# B&R Automation Studio project JOB_NUMBER (part 5)

#### Kan_Driver.ab
```automation-basic
(********************************************************************
 * COPYRIGHT -- HP
 ********************************************************************
 * Program: Kan_Driver
 * File: Kan_Driver.ab
 * Author: treamsbottom
 * Created: September 07, 2012
 ********************************************************************
 * Implementation of program Kan_Driver
 ********************************************************************)
;----------------------------------------------------------------------------------------------------------------;
;-----21-1-2013..TR..Version A6 - First TestedVersion - Note 2 Specials in overview clien to run with Shuttle
;-----28-1-2013..TR..Version A7 - Remove Specials..Add option to send program and category number & Batch number.
;-----20-5-2014..TR..Version A12 - Fix ValidCat on DataValid
;-----09-01-2015..TR..Version A14 - Add Batching control
;-----02-08-2016 ..TR..Version A17 - Add Syncronous loading to Server Cmd 1000.. Use Comm[x].Transfer to watch for permission to unload.
;-----03-03-2017..TR.Version A18 - Add "Advanced Connection Mode"
;-----07-06-2017 ..TR..Version A19 - Fix issues with sending empty bag date-- Remove reference to Comm[].Category -- Read all information from bag for consistency.
;-----24-07-2018 ..TR -- Versioning Stopped Issues now tracked in GIT.
;-----------------------------------------------------------------------------------------------------------------
PROGRAM _INIT
	comm ACCESS ADR(Comm[0]);
END_PROGRAM
PROGRAM _CYCLIC
;Monitor State of supertrack (only send basic states now).
;IF (Kanlink.Server.Enable OR Kanlink.Client.Enable OR Kanlink.OverviewClient.Enable OR Kanlink.OverviewServer.Enable) THEN
;	IF SafetyZone[1].HaltSys THEN
;		SuperTrackState = KG_MACHINESTATE_EMERGENCYSTOP
;	ELSE
;		SuperTrackState = KG_MACHINESTATE_AUTOMATIC_RUN
;	ENDIF
;ENDIF
;--------------------------------------------------Kanlink Server Communication-----------------------------------------------------------------
IF Kanlink.Server.Enable THEN
	;Populate Batch Data
	LOOP n = 1 TO Kanlink.Server.MaxConns  DO
		IF (Kanlink.Server.IP[n].Adr > 0) THEN
			LOOP Index = 1 TO 1 DO ; Loop through each bag buffer
				comm ACCESS ADR(Comm[Kanlink.Server.IP[n].CommID]);
				IF (comm.Category > 0) THEN
					GetTimeStamp.enable = 1
					GetTimeStamp FUB DTGetTime()
					Batch[n].BatchData[Index].dtTimeStamp = GetTimeStamp.DT1
					;Make a string out OF CAT AND CUS
					length = itoa(comm.Category,ADR(myCategoryString));
					length = itoa(comm.Customer,ADR(myCustomerString));
					;copy Bag Data to KanLink Bag data type
;					IF Kanlink.GlobalSettings.TransferProgramCode THEN
;						Batch[n].BatchData[Index].sCategory = myProgramString
;						length = memcpy(ADR(Batch[n].BatchData[Index].bCustom),ADR(myCategoryString),12)
;					ELSE IF Kanlink.GlobalSettings.TransferProgin_bCustom THEN
;						Batch[n].BatchData[Index].sCategory = myCategoryString
;						length = memcpy(ADR(Batch[n].BatchData[Index].bCustom),ADR(myProgramString),12)
;					ELSE
						Batch[n].BatchData[Index].sCategory = myCategoryString
;					ENDIF
					IF Kanlink.GlobalSettings.UseBatchCode THEN
						IF Kanlink.GlobalSettings.BatchCodeTyp = BatchTyp_UDINT THEN
							;length = itoa(Bag[BagNumber].Mis,ADR(Batch[n].BatchData[Index].bBatchNo)) ; Convert to string
							length = memcpy(ADR(Batch[n].BatchData[Index].bBatchNo),ADR(comm.BatchID),4) ; Direct UDINT copy unreadble in KANLINK data.
						ELSE IF Kanlink.GlobalSettings.BatchCodeTyp = BatchTyp_16Byte THEN
							;Bag typ does not support this yet..
						ENDIF
					ELSE
						length = strcpy(ADR(Batch[n].BatchData[Index].bBatchNo),"")
					ENDIF
					Batch[n].BatchData[Index].bCntCustomers = 1
					Batch[n].BatchData[Index].wTotalWeight = comm.Weight;Summary weight of all Part Customers in the Bag, normally 1
					;First Customer in the Bag

					IF (comm.Batch_QtyRemaining <= 1) THEN
						Batch[n].BatchData[Index].PartBatch[0].sCustomNo = myCustomerString
						Batch[n].BatchData[Index].PartBatch[0].wCustomWeight = comm.Weight;Bag[BagNumber].Wgt
					ELSE
						Batch[n].BatchData[Index].bCntCustomers = USINT(comm.Batch_QtyRemaining)
						LOOP t = 0 TO 7 DO
							length = itoa(comm.Batchpart[t].Customer,ADR(myCustomerString));
							Batch[n].BatchData[Index].PartBatch[t].sCustomNo = myCustomerString
							Batch[n].BatchData[Index].PartBatch[t].wCustomWeight = comm.Batchpart[t].Wgt
						ENDLOOP
					ENDIF
				ELSE
					strcpy(ADR(myCategoryString),ADR(""));
					strcpy(ADR(myCustomerString),ADR(""))
					strcpy(ADR(myProgramString),ADR(""));
					Batch[n].BatchData[Index].bCntCustomers = 0
					Batch[n].BatchData[Index].sCategory = myCategoryString
					length = strcpy(ADR(Batch[n].BatchData[Index].bCustom),"")
					length = strcpy(ADR(Batch[n].BatchData[Index].bBatchNo),"")
					Batch[n].BatchData[Index].wTotalWeight = 0 ;Summaray weight of all Part Customers in the Bag, normally 1
					LOOP t = 0 TO 7 DO
						Batch[n].BatchData[Index].PartBatch[t].sCustomNo = myCustomerString
						Batch[n].BatchData[Index].PartBatch[t].wCustomWeight = 0
					ENDLOOP
				ENDIF
				PT100[n].Resp.BatchData = Batch[n].BatchData[1] ; Only send first bag over KANLINK
			ENDLOOP

			; Handshake Signal Convert Comm into the KANLINK protocol
			;ValidCat = 	strcmp(ADR(comm.Category), "")
			//BagNumber = Kanlink.Server.BagNum[n].BagNums[1];
			IF (comm.Category > 0) THEN
				PT100[n].Resp.xHsDataValid = TRUE;
			ELSE
				PT100[n].Resp.xHsDataValid = FALSE
				PT100[n].Resp.xHsUnloading = FALSE
			ENDIF

			IF comm.BagReady THEN
				PT100[n].Resp.xHsReqForUnload = TRUE;
			ELSE
				PT100[n].Resp.xHsReqForUnload = FALSE;
			ENDIF

			comm.ReadyToLoad	= PT100[n].Req.xHready;
			comm.DropLoad 		= PT100[n].Req.xHreadyForLoad;
			comm.LoadDropped  	= PT100[n].Req.xHbatchReceived;
			PT100[n].Resp.wCntLoads = comm.Batch_QtyRemaining

			IF comm.DropLoad THEN
				PT100[n].Resp.xHsUnloading = TRUE
			ENDIF

			IF comm.HaltSys THEN
				PT100[n].Resp.wState = KG_MACHINESTATE_EMERGENCYSTOP
			ELSE
				PT100[n].Resp.wState = KG_MACHINESTATEX_AUTOMATIC_RUN
			ENDIF

			comm.Live = IFhlKanLink.Server[n].out.xConnected
		;Syncronous Loading.
			IF PT100[n].Req.xHreqCtrlTransfer THEN
				//Syncronous loading. Only allow unload when bit .x.x.x. is on
				PT100[n].Resp.xHsTransferRunning := PT100[n].Req.xHwaitingForTransfer;
			ELSE
				//Always give permission to unload..
				PT100[n].Resp.xHsTransferRunning := 1;
			ENDIF;
			comm.Transfer := PT100[n].Resp.xHsTransferRunning
		ENDIF
	ENDLOOP
ENDIF//ServerDriver
;--------------------------------------------------------Client Driver------------------------------------------------------------------
IF Kanlink.Client.Enable THEN
	LOOP n = 1 TO Kanlink.Client.MaxConns DO
		comm  ACCESS ADR(Comm[Kanlink.Client.IP[n].CommID])
		;Give Machine Ready
		PTResp[n].Req.xHready = TRUE
		PTResp[n].Req.bHcmdAutomatic = TRUE

		comm.BagReady = PTResp[n].Resp.xHsReqForUnload
		;Give ready to load when Ready
		PTResp[n].Req.xHreadyForLoad = comm.ReadyToLoad
		PTResp[n].Req.xHtransferRunning = comm.Transfer

		PTResp[n].Req.xHbatchReceived = comm.LoadRecieved
			;Send supertrack state
		IF comm.HaltSys THEN
			PTResp[n].Req.wHstate = KG_MACHINESTATE_EMERGENCYSTOP
		ELSE
			PTResp[n].Req.wHstate = KG_MACHINESTATEX_AUTOMATIC_RUN
		ENDIF
		;Check for Data Valid and unloading start.	then copy data to Comm Variable
		UnloadingPulse[n].CLK = (PTResp[n].Resp.xHsUnloading AND PTResp[n].Resp.xHsDataValid)
		UnloadingPulse[n] FUB R_TRIG()
		IF UnloadingPulse[n].Q THEN
;			IF Kanlink.GlobalSettings.TransferProgramCode THEN
;				comm.Program = USINT(atoi(ADR(PTResp[n].Resp.BatchData.sCategory)))
;				comm.Category = atoi(ADR(PTResp[n].Resp.BatchData.bCustom))
;			ELSE IF Kanlink.GlobalSettings.TransferProgin_bCustom THEN
;				comm.Program = USINT(atoi(ADR(PTResp[n].Resp.BatchData.bCustom)))
;				comm.Category = atoi(ADR(PTResp[n].Resp.BatchData.sCategory))
;			ELSE
				comm.Category = atoi(ADR(PTResp[n].Resp.BatchData.sCategory))
;			ENDIF
			comm.Customer = atoi(ADR(PTResp[n].Resp.BatchData.PartBatch[0].sCustomNo))
			comm.Weight = PTResp[n].Resp.BatchData.wTotalWeight
			IF Kanlink.GlobalSettings.UseBatchCode THEN
				IF Kanlink.GlobalSettings.BatchCodeTyp = BatchTyp_UDINT THEN
					length = memcpy(ADR(comm.BatchID),ADR(PTResp[n].Resp.BatchData.bBatchNo),4)
				ELSE IF Kanlink.GlobalSettings.BatchCodeTyp = BatchTyp_16Byte THEN
					;Bag typ does not support this yet..
				ENDIF
			ELSE
				comm.BatchID = 0
			ENDIF
		ENDIF

		comm.Unloading =  PTResp[n].Resp.xHsUnloading
		UnloadingFinishPLS[n].CLK = PTResp[n].Resp.xHsUnloading
		UnloadingFinishPLS[n] FUB F_TRIG()

		comm.UnloadFinished = UnloadingFinishPLS[n].Q
		;Comm Live
		comm.Live = IFhlKanLink.Client[n].out.xConnected
	ENDLOOP
ENDIF
;;---------------------------------------------------------------------------------------------Overview Client----------------------------------------
;IF Kanlink.OverviewClient.Enable THEN ; Collect data
;;------------------------------------------Build Request---------------------------------------------------
;
;	LOOP n = 1 TO Kanlink.OverviewClient.MaxConns DO
;
;
;		IF (CANOffset > 0) THEN
;			CANOffset = (Kanlink.OverviewClient.CANOffset - 1)
;			Comm[n+CANOffset].Live = IFhlKanLink.Client[n+Kanlink.OverviewClient.IndexOffset].out.xConnected
;			IF NOT Comm[n+CANOffset].Live THEN
;				D[Kanlink.OverviewClient.StatusReg[n]] = 0
;			ENDIF
;		ELSE
;			CANOffset = 0
;		ENDIF;
;
;		IF Kanlink.OverviewClient.InfoReq[n].wNoOfPosition[6] = 0 THEN ; do not multiplex data.
;			STOverReq[n].Req.wCntPositions = Kanlink.OverviewClient.InfoReq[n].wCntPositions;Number of Bags requested
;			DataOffset[n] = 0
;		ELSE
;
;			DataCount = 0
;			LOOP x = 0 TO 5 DO
;				IF (STOverReq[n].Req.wNoOfPosition[x] > 0) THEN
;					DataCount = DataCount + 1
;				ENDIF
;				IF DataCount > 5 THEN
;					DataCount = 6
;				ENDIF
;			ENDLOOP
;			STOverReq[n].Req.wCntPositions = DataCount;Number of Bags requested
;		ENDIF
;
;
;		LOOP x = 0 TO 5 DO
;			;datapositions requested
;			EXITIF ((DataOffset[n] + x) > HLKANLINK_MAX_OVERVIEW_DATA)
;
;			STOverReq[n].Req.wNoOfPosition[x] = Kanlink.OverviewClient.InfoReq[n].wNoOfPosition[x + DataOffset[n]]
;				;-----------------------------------------------Read Data----------------------------------
;			IF (STOverReq[n].Resp.wNoOfPositions[x] > 0) AND ((x <= STOverReq[n].Resp.wCntPositions) OR (STOverReq[n].Resp.wCntPositions = 0 )) THEN
;				IF (Kanlink.OverviewClient.InfoResp[n].BagNum[x + DataOffset[n]] > 0) THEN
;					IF Kanlink.OverviewClient.InfoReq[n].wNoOfPosition[x+DataOffset[n]] = STOverReq[n].Resp.wNoOfPositions[x] THEN
;					//	D[Kanlink.OverviewClient.StatusReg[n]] = STOverReq[n].Resp.wMachineState
;						BagIndex = Kanlink.OverviewClient.InfoResp[n].BagNum[x + DataOffset[n]]
;						IF Kanlink.GlobalSettings.TransferProgramCode THEN
;							Bag[BagIndex].Prg = USINT(atoi(ADR(STOverReq[n].Resp.BatchData[x].sCategory)))
;							Bag[BagIndex].Cat = atoi(ADR(STOverReq[n].Resp.BatchData[x].bCustom))
;						ELSE IF Kanlink.GlobalSettings.TransferProgin_bCustom THEN
;							Bag[BagIndex].Prg = USINT(atoi(ADR(STOverReq[n].Resp.BatchData[x].bCustom)))
;							Bag[BagIndex].Cat = atoi(ADR(STOverReq[n].Resp.BatchData[x].sCategory))
;						ELSE
;							Bag[BagIndex].Cat = atoi(ADR(STOverReq[n].Resp.BatchData[x].sCategory))
;						ENDIF
;						Bag[BagIndex].Cus = atoi(ADR(STOverReq[n].Resp.BatchData[x].PartBatch[0].sCustomNo)) ; Standard line of code..
;						Bag[BagIndex].Wgt = STOverReq[n].Resp.BatchData[x].PartBatch[0].wCustomWeight
;						IF Kanlink.GlobalSettings.UseBatchCode THEN
;							IF Kanlink.GlobalSettings.BatchCodeTyp = BatchTyp_UDINT THEN
;									length = memcpy(ADR(Bag[BagIndex].Mis),ADR(STOverReq[n].Resp.BatchData[x].bBatchNo),4)
;								ELSE IF	Kanlink.GlobalSettings.BatchCodeTyp = BatchTyp_16Byte THEN
;								;Not supported yet....
;							ENDIF
;						ELSE
;							Bag[BagIndex].Mis = 0
;						ENDIF
;					ENDIF
;				ENDIF
;			ENDIF
;		ENDLOOP
;		IF STOverReq[n].Resp.wNoOfPositions[0] = Kanlink.OverviewClient.InfoReq[n].wNoOfPosition[DataOffset[n]] THEN
;			DataOffset[n] = DataOffset[n] + 6
;		ELSE IF Kanlink.OverviewClient.InfoReq[n].wNoOfPosition[DataOffset[n]] = 0 THEN
;			DataOffset[n] = 0
;		ENDIF
;	ENDLOOP
;ENDIF
;
;;---------------------------------------------------------------------------------------------Overview Server----------------------------------------
;IF Kanlink.OverviewServer.Enable THEN
;	LOOP n = 1 TO Kanlink.OverviewServer.MaxConns DO
;		IF (STOverResp[n].Req.wCntPositions <= 6) THEN
;			IF (STOverResp[n].Req.wCntPositions = 0) OR (STOverResp[n].Req.wCntPositions = 6) THEN
;				NoOfDataRequested = 5
;			ELSE
;				NoOfDataRequested = STOverResp[n].Req.wCntPositions
;			ENDIF
;			LOOP x = 0 TO 5 DO
;				IF x <= NoOfDataRequested THEN
;					BagIndex = STOverResp[n].Req.wNoOfPosition[x]
;
;					//STOverResp[n].Resp.wMachineState = SuperTrackState
;					STOverResp[n].Resp.wNoOfPositions[x] = BagIndex
;					STOverResp[n].Resp.wCntPositions = 	STOverResp[n].Req.wCntPositions
;					itoa(Bag[BagIndex].Prg,ADR(sProgram))
;					itoa(Bag[BagIndex].Cat,ADR(sCategory))
;					itoa(Bag[BagIndex].Cus,ADR(sCustomer))
;					itoa(Bag[BagIndex].Mis,ADR(sBatchID))
;					STOverResp[n].Resp.BatchData[x].dtTimeStamp = GetTimeStamp.DT1
;					IF Kanlink.GlobalSettings.TransferProgramCode THEN
;						strcpy(ADR(STOverResp[n].Resp.BatchData[x].sCategory),ADR(sProgram))
;						strcpy(ADR(STOverResp[n].Resp.BatchData[x].bCustom),ADR(sCategory))
;					ELSE IF Kanlink.GlobalSettings.TransferProgin_bCustom THEN
;						strcpy(ADR(STOverResp[n].Resp.BatchData[x].sCategory),ADR(sCategory))
;						strcpy(ADR(STOverResp[n].Resp.BatchData[x].bCustom),ADR(sProgram))
;					ELSE
;						strcpy(ADR(STOverResp[n].Resp.BatchData[x].sCategory),ADR(sCategory))
;					ENDIF
;					IF Kanlink.GlobalSettings.UseBatchCode THEN
;						IF Kanlink.GlobalSettings.BatchCodeTyp = BatchTyp_UDINT THEN
;							length = memcpy(ADR(STOverResp[n].Resp.BatchData[x].bBatchNo),ADR(Bag[BagIndex].Mis),4)
;						ELSE IF Kanlink.GlobalSettings.BatchCodeTyp = BatchTyp_UDINT THEN
;							strcpy(ADR(STOverResp[n].Resp.BatchData[x].bBatchNo),ADR(sBatchID))
;						ENDIF
;					ELSE
;						strcpy(ADR(STOverResp[n].Resp.BatchData[x].bBatchNo),"")
;					ENDIF
;					strcpy(ADR(STOverResp[n].Resp.BatchData[x].PartBatch[0].sCustomNo),ADR(sCustomer))
;					STOverResp[n].Resp.BatchData[x].PartBatch[0].wCustomWeight = Bag[BagIndex].Wgt
;				ELSE
;					STOverResp[n].Resp.wNoOfPositions[x] = 0
;					STOverResp[n].Resp.BatchData[x].dtTimeStamp = 0
;					strcpy(ADR(STOverResp[n].Resp.BatchData[x].sCategory),"")
;					strcpy(ADR(STOverResp[n].Resp.BatchData[x].bCustom),"")
;					strcpy(ADR(STOverResp[n].Resp.BatchData[x].bBatchNo),"")
;					strcpy(ADR(STOverResp[n].Resp.BatchData[x].PartBatch[0].sCustomNo),"")
;					STOverResp[n].Resp.BatchData[x].PartBatch[0].wCustomWeight = 0
;				ENDIF
;			ENDLOOP
;		ENDIF
;	ENDLOOP
;ENDIF

END_PROGRAM
```

### Package Logical/Standard/Kanlink/CAN - CAN Communication Variables

### CAN.typ
```iecst
TYPE
	WET_CAN : 	STRUCT
		ControlSignals : USINT;
		ControlSignals2 : USINT;
		Category : UINT;
		Customer : UINT;
		Weight : UINT;
	END_STRUCT;
	DRY_CAN : 	STRUCT
		ControlSignals : USINT;
		ControlByte2 : USINT;
		Category : UDINT;
		Weight : UINT;
	END_STRUCT;
	DRY_CAN1 : 	STRUCT
		CustomerCode : UDINT;
		BatchCode : UDINT;
	END_STRUCT;
	DRYCAN_comm_typ : 	STRUCT
		ReadFrame : DRY_CAN;
		WriteFrame : DRY_CAN;
		WriteFrame1 : DRY_CAN1;
		EventRead : BOOL;
		EventWrite : BOOL;
		EventWrite1 : BOOL;
	END_STRUCT;
	Comm_typ : 	STRUCT
		StrobeComplete : BOOL;
		BagReady : BOOL;
		BatchCode : UINT;
		Category : UDINT;
		Customer : UDINT;
		Destination : UINT;
		DropLoad : BOOL;
		DoubleLoad : BOOL;
		Live : BOOL;
		LiveTime : UINT;
		LoadDropped : BOOL;
		LoadFinished : BOOL;
		Program : UINT;
		ReadyToLoad : BOOL;
		UnloadFinished : BOOL;
		Weight : UINT;
		BatchID : UDINT;
		Batch_QtyRemaining : UINT;
		LoadRecieved : BOOL;
		Unloading : BOOL;
		Batchpart : ARRAY[0..7]OF Batchpart_typ;
		Batchpart_wgt : ARRAY[0..9]OF UINT;
		Count : UINT;
		Bid : UDINT; (**Internal use only pass bid ID>*)
		TimeStamp : DATE_AND_TIME; (**Internal use only*)
		Transfer : BOOL;
		HaltSys : BOOL;
	END_STRUCT;
	Batchpart_typ : 	STRUCT
		Wgt : UINT;
		Customer : UDINT;
	END_STRUCT;
END_TYPE
```

### CAN.var
```iecst
VAR CONSTANT
	MAX_COMM : USINT := 30;
END_VAR
VAR
	Comm : ARRAY[0..MAX_COMM] OF Comm_typ;
END_VAR
VAR CONSTANT
	COMM_CLEAR : Comm_typ := (0);
END_VAR
```

### Program Logical/Standard/Kanlink/kanlink_map (IEC) - *Custom task to convert Kanlink PLC to eVue Comms

#### Variables.var
```iecst
VAR
	bag_2_wieight : INT;
	doubleDrop : BOOL;
	DryerOpenTimer1 : TON;
	DryerOpenTimer2 : TON;
	DryerOpenTimer3 : TON;
	DryerOpenTimer4 : TON;
	DryerOpenTimer5 : TON;
	DryerOpenTimer6 : TON;
	DryerOpenTimer7 : TON;
	DryerOpenTimer8 : TON;
	DryerOpenTimer9 : TON;
	DryerOpenTimer10 : TON;
	DryerOpenTimer11 : TON;
	DryerOpenTimer12 : TON;
	DryerOpenTimer13 : TON;
	DryerOpenTimer14 : TON;
	DryerOpenTimer15 : TON;
	DryerOpenTimer16 : TON;
	WasherOpenTimer1 : TON;
	WasherOpenTimer2 : TON;
	WasherOpenTimer3 : TON;
	WasherOpenTimer4 : TON;
	WasherOpenTimer5 : TON;
	WasherOpenTimer6 : TON;
	WasherOpenTimer7 : TON;
	WasherOpenTimer8 : TON;
	WasherOpenTimer9 : TON;
	WasherOpenTimer10 : TON;
END_VAR
```

#### Cyclic.st
```iecst
PROGRAM _CYCLIC
//	//Opener code
//
//
//	//Tunnel X
//	r56.open_signal	:= 	Comm[1].DropLoad;
//	r56.receive_signal	:= 	Comm[1].LoadDropped;
//	Comm[1].BagReady	:= r56.sling_ready;
//
//	IF r56.sling_ready THEN
//		Comm[1].Customer	:= wash_com_cust_1;
//		Comm[1].Category	:= wash_com_cat_1;
//		Comm[1].BatchID		:= DByte_TO_4Byte(ADR(wash_com_batch1_1),ADR(wash_com_batch2_1));
//		Comm[1].Weight		:= (wash_com_wt_1 * 10);
//	ELSE
//		Comm[1].Customer	:= 0;
//		Comm[1].Category	:= 0;
//		Comm[1].BatchID		:= 0;
//		Comm[1].Weight		:= 0;
//	END_IF;
//
//	IF EDGEPOS(r56.fire) THEN
//		wash_com_cust_1 := 0;
//		wash_com_cat_1  := 0;
//		wash_com_wt_1  := 0;
//		wash_com_batch1_1 := 0;
//		wash_com_batch2_1 := 0;
//	END_IF;
//
//
//
//
//	//Washer X
//	WasherOpenTimer1(IN:= r60.sling_ready AND Comm[3].DropLoad, PT := t#1500ms);
//	IF EDGEPOS(Comm[3].ReadyToLoad) THEN
//		r60.transfer_requested_signal := TRUE;
//	END_IF;
//
//	r60.open_signal	:= 	WasherOpenTimer1.Q;
//	r60.receive_signal	:= 	Comm[3].LoadDropped;
//	Comm[3].BagReady	:= r60.sling_ready;
//
//
//	IF r60.sling_ready THEN
//		Comm[3].Customer	:= wash_com_cust_3;
//		Comm[3].Category	:= wash_com_cat_3;
//		Comm[3].BatchID		:= DByte_TO_4Byte(ADR(wash_com_batch1_3),ADR(wash_com_batch2_3));
//		Comm[3].Weight		:= (wash_com_wt_3 * 10);
//	ELSE
//		Comm[3].Customer	:= 0;
//		Comm[3].Category	:= 0;
//		Comm[3].BatchID		:= 0;
//		Comm[3].Weight		:= 0;
//	END_IF;
//
//	IF EDGEPOS(r60.fire) OR NOT(Comm[3].ReadyToLoad) THEN
//		r60.transfer_requested_signal := FALSE;
//	END_IF;
//
//	IF EDGEPOS(r60.fire) THEN
//		wash_com_cust_3 := 0;
//		wash_com_cat_3  := 0;
//		wash_com_wt_3  := 0;
//		wash_com_batch1_3 := 0;
//		wash_com_batch2_3 := 0;
//	END_IF;
//
//
//
//	//Dryer X
//	DryerOpenTimer1(IN:= r106.sling_ready AND Comm[6].DropLoad, PT := t#1500ms);
//	r106.transfer_requested_signal := Comm[6].ReadyToLoad;
//	r106.open_signal	:= 	DryerOpenTimer1.Q;
//	r106.receive_signal	:= 	Comm[6].LoadDropped;
//	Comm[6].BagReady	:= r106.sling_ready;
//
//	IF r106.sling_ready THEN
//		Comm[6].Customer	:= wash_com_cust_10;
//		Comm[6].Category	:= wash_com_cat_10;
//		Comm[6].BatchID		:= DByte_TO_4Byte(ADR(wash_com_batch1_10),ADR(wash_com_batch2_10));
//		Comm[6].Weight		:= (wash_com_wt_10 * 10);
//	ELSE
//		Comm[6].Customer	:= 0;
//		Comm[6].Category	:= 0;
//		Comm[6].BatchID		:= 0;
//		Comm[6].Weight		:= 0;
//	END_IF;
//
//	IF EDGEPOS(r106.fire) THEN
//		wash_com_cust_10 := 0;
//		wash_com_cat_10  := 0;
//		wash_com_wt_10  := 0;
//		wash_com_batch1_10 := 0;
//		wash_com_batch2_10 := 0;
//	END_IF;
//
//
//
//
//
//
//	// Transfers
//
//	//Wet Transfer X
//	wash_com_cust_6 	:= UDINT_TO_INT(Comm[28].Customer);
//	wash_com_cat_6 		:= UDINT_TO_INT(Comm[28].Category);
//	wash_com_wt_6 		:= (Comm[28].Weight/10);
//	wash_com_batch1_6	:= Get_Lower2Bytes(Comm[28].BatchID);
//	wash_com_batch2_6	:= Get_Higher2Bytes(Comm[28].BatchID);
//	//	Comm[28].bCustom[0]
//
//
//	Comm[28].ReadyToLoad	:= r80.sling_ready;
//	r80.transfer_requested_signal := Comm[28].BagReady;
//	r80.xfer_in_progress	:= Comm[28].Unloading;
//	r80.xfer_complete := Comm[28].UnloadFinished;
//
//	IF EDGEPOS(r80.fire) THEN
//		wash_com_cust_6 := 0;
//		wash_com_cat_6 := 0;
//		wash_com_wt_6 := 0;
//		wash_com_batch1_6 := 0;
//		wash_com_batch2_6 := 0;
//	END_IF;
END_PROGRAM
```

### Package Logical/Standard/Kanlink/KGFramework - Standard-Packages

### Package Logical/Standard/Kanlink/KGFramework/Pkg_KGStandard - Kannegiesser Standards

### Library Logical/Standard/Kanlink/KGFramework/Pkg_KGStandard/KGstdLib (IEC) - Kannegiesser Hilfsfunktionen
Depends on: astime, AsIODiag, Ethernet, AsBrStr, DataObj, AsArLog

#### kgGetEthPort.st - Returns the CPUs ethernet port as string
```iecst
(********************************************************************
* COPYRIGHT -- Microsoft
********************************************************************
* Library: Netlink
* File: GetEthPort.st
* Author: hunholz
* Created: June 30, 2011
********************************************************************
* Implementation of library Netlink
********************************************************************)

(* Returns the CPUs ethernet port as string *)
FUNCTION_BLOCK kgGetEthPort

IF enable THEN

	IF adrIF <= 16#3FFF THEN

		_bStep := 10;
		status := KG_ERR_GETETHPORT_ADRIF;
		RETURN;

	END_IF

	_xReady := FALSE;

	REPEAT

		CASE (_bStep) OF

			10:
				// Create Info
					DiagCreateInfo_CPU(enable := TRUE, infoKind := asdiagPLUGGED);

					status := DiagCreateInfo_CPU.status;

					IF (status = ERR_OK) THEN
			  			_bStep := 12;
					END_IF;

				12:
					// Get Info
					DiagGetNumInfo_CPU(enable := TRUE,
											ident := DiagCreateInfo_CPU.ident,
											index := 0,
											infoCode := asdiagPLUGGED_MODNO);

					status := DiagGetNumInfo_CPU.status;

					IF (status = ERR_OK) THEN

						CASE DiagGetNumInfo_CPU.value OF

							KG_CPU_X20CP1484, KG_CPU_X20CP1484_1, KG_CPU_X20CP3484_1, KG_CPU_X20CP1486, KG_CPU_X20CP3486, KG_CPU_X20CP3585, KG_CPU_X20CP1584,KG_CPU_X20CP1586, KG_CPU_X20CP3484:
								brsstrcpy(adrIF, ADR('IF2'));

							KG_CPU_PP420_1043_75, KG_CPU_CTT_11, KG_CPU_PP65_0571_P74, KG_CPU_PCT_04, KG_CPU_PCT_03:
								brsstrcpy(adrIF, ADR('IF5'));

							ELSE	// keinen gültigen B&R ID-Code gefunden
								brsstrcpy(adrIF, ADR('IF3'));
								//status := KG_ERR_GETETHPORT_IFSTRING;

						END_CASE

					_bStep := 14;

					ELSIF (status <> ERR_FUB_BUSY) THEN
						_bStep := 10;
				END_IF;

			14:
				 //Write string TO variable

				DiagDisposeInfo_CPU(enable := TRUE, ident := DiagCreateInfo_CPU.ident);

				status := DiagDisposeInfo_CPU.status;

				_xReady := (status = ERR_OK);

				IF (status <> ERR_FUB_BUSY) THEN

					_bStep := 10;
					DiagCreateInfo_CPU(enable := FALSE);
					DiagDisposeInfo_CPU(enable := FALSE);
					DiagGetNumInfo_CPU(enable := FALSE);

				END_IF;

			ELSE

				_bStep := 10;
				status := ERR_FUB_BUSY;

		END_CASE;

		UNTIL

		status <> ERR_OK OR _xReady

	END_REPEAT

ELSE

	status := ERR_FUB_ENABLE_FALSE;
	_bStep := 10;

END_IF

END_FUNCTION_BLOCK
```


- Program Logical/Standard/Kanlink/KGFramework/Pkg_mnSystem/mnSystem (IEC) - Systemtask für Versionierung (no source held here)

- Program Logical/Standard/Kanlink/KGFramework/Pkg_mnEth/mnEth (IEC) - Ethernetmanager (no source held here)

- Program Logical/Standard/Kanlink/KGFramework/Pkg_mnCnt/mnCnt (IEC) - Counter Manager (no source held here)

- Program Logical/Standard/Kanlink/KGFramework/Pkg_mnMsg/mnMsg (IEC) - Meldungsmanager (no source held here)

- Library Logical/Standard/Kanlink/KGFramework/Pkg_mnMsg/KGlibMsg (IEC) - A new source library (no source held here)

### Package Logical/Standard/Kanlink/KGFramework/Pkg_mnParam - Parameter-Manager

- Program Logical/Standard/Kanlink/KGFramework/Pkg_mnParam/mnParam (IEC) - Parameter Manager (no source held here)

### Library Logical/Standard/Kanlink/KGFramework/Pkg_mnParam/mnParamLib (IEC)
Depends on: astime


- Program Logical/Standard/Kanlink/KGFramework/Pkg_mnTxt/mnTxt (IEC) - Text-Manager (no source held here)

- Program Logical/Standard/Kanlink/KGFramework/Pkg_hlDFII/hlDFII (IEC) - Statemachine zur Abfrage einer SQL-Datenbank (no source held here)

- Program Logical/Standard/Kanlink/KGFramework/Pkg_mnTest/mnTest (IEC) - Testadapter (no source held here)

- Program Logical/Standard/Kanlink/KGFramework/Pkg_svCPCache/svCPCache (IEC) - Category-Program-Cache (no source held here)

### Program Logical/Standard/Kanlink/KGFramework/Pkg_hlKanLink/hlKanLink (IEC) - Kanlink Task

#### KanLinkCyclic.st - Cyclic code
```iecst
(********************************************************************
 * COPYRIGHT -- Herbert Kannegiesser GmbH
 ********************************************************************
 * Program: KanLink
 * File: KanLinkCyclic.st
 * Author: stahlhut
 * Created: December 23, 2011
 ********************************************************************
 * Implementation of program WetLink
 ********************************************************************)

(*

	Falls ohne Framework gearbeitet werden soll in den Eigenschaften der Task hlKanLink (Config. View Cpu.sw)
	im Tab. Compiler im Feld "Additional build options:" -D HLKANLINK_AUTONOM  eintragen
	Dazu das Package KanLinkAutonom importieren

*)

PROGRAM _CYCLIC

// Struktur für Visualisierung füllen

IFhlKL_Visu.out.iCycleTime := Kanlink._iCycleTime;
IFhlKL_Visu.out.step := Kanlink.Step;
IFhlKL_Visu.out.udNetId := Kanlink.udNetID;
IFhlKL_Visu.out.udpOpenStatus := Kanlink.udp.open.status;
IFhlKL_Visu.out.udpRecStatus := Kanlink.udp.rec.status;
IFhlKL_Visu.out.udpSendStatus := Kanlink.udp.send.status;
_wClt := LIMIT(0,IFhlKL_Visu.in.iCltNr,HLKANLINK_MAX_CLIENTCONNS);
  _wSrv := LIMIT(0,IFhlKL_Visu.in.iServerNr,HLKANLINK_MAX_SERVERCONNS);
IFhlKL_Visu.out.client := Kanlink.ClientListe[_wClt];
IFhlKL_Visu.out.server := Kanlink.ServerListe[_wSrv];

// Commando von der Visu verarbeiten
// Commando nur setzen wenn CmdResp = 0
// aufrufer muss nach ausführung cmdNr wieder auf 0 setzen!
IF IFhlKL_Visu.in.cmdNr <> IFhlKL_Visu.out.cmdResp THEN
	CASE IFhlKL_Visu.in.cmdNr OF
		0: IFhlKL_Visu.out.cmdResp := 0;
		1: // Neustart
			IFhlKL_Visu.out.cmdResp := 1;
			Kanlink.Step := 1;
		2: // Neustart mit lastId = 1
			Kanlink._uiLastId := 1;
			IFhlKL_Visu.out.cmdResp := 1;
			Kanlink.Step := 2;
		ELSE
			// unbekanntes Commando
			IFhlKL_Visu.out.cmdResp := 16#7FFF;

	END_CASE;
END_IF;

#ifndef HLKANLINK_AUTONOM // Logging nur mit kg-Framework

	// ===========================
	// Logging
	// ===========================

	IF _xRBReady THEN

		CASE _wLogStep OF

			0:
				_ReadRB(wPtrRead := _wPtrRBread, wPtrStart := _wPtrRBstart, wPtrWrite := _wPtrRBwrite);

				IF _ReadRB.wStatus = ERR_OK THEN

					CASE _LogEntry.wErrorNo OF

						0:
							_kgArLogWrite.text := 'OK';

						HLKANLINK_MSG_NO_STRUCDEF:

							_kgArLogWrite.text := 'Create Strucdefinition failed : {##AttrVar1} / {##AttrVar2}';
							_kgArLogWrite.var1 := _LogEntry.lAttr1;

						ELSE

							_kgArLogWrite.text := UINT_TO_STRING(_LogEntry.wErrorNo);
							_kgArLogWrite.text := CONCAT(_kgArLogWrite.text, ' : {##AttrVar1} / {##AttrVar2}');
							_kgArLogWrite.var1 := _LogEntry.lAttr1;
							_kgArLogWrite.var2 := _LogEntry.lAttr2;

					END_CASE

					_wLogStep := 1;

				END_IF

			1:
				_kgArLogWrite();

				IF _kgArLogWrite.status <> ERR_FUB_BUSY THEN

					_wLogStep := 0;

				END_IF

		END_CASE

	END_IF

	IF _wDebIdx >= 0 AND _wDebIdx <= _HLKANLINK_MAX_IDX_DEFSTRUC THEN

		IF _lPtrStrucDef[_wDebIdx] > 0 THEN

			_sDebString ACCESS _lPtrStrucDef[_wDebIdx] + _wDebOffset;

		END_IF

	END_IF

#endif

	// =======================================================================

	IF _xInitOK THEN

		IF _xSaveConfig THEN
			KL_SaveConfDO_0(adrName :=ADR('KL_Conf') , adrDaten := ADR(IFhlKanLink.Parameter), len := SIZEOF( IFhlKanLink.Parameter));
			IF KL_SaveConfDO_0.status <> ERR_FUB_BUSY THEN // fertig
				_xSaveConfig := FALSE;
			END_IF;
		END_IF;

		IF EDGEPOS(IFhlKanLink.in.xRun ) THEN
			IF Kanlink.Step = 0 THEN
				Kanlink.Step := 1;
			END_IF;
		END_IF;
		IF EDGENEG(IFhlKanLink.in.xRun) THEN // stoppen
			IF Kanlink.Step <> 0 THEN
				Kanlink.Step := 20;
			END_IF;
		END_IF;

		IF IFhlKanLink.in.xRestart THEN
			Kanlink.Step := 1;
			IFhlKanLink.in.xRestart := 0;
		END_IF;

		IFhlKanLink.xError := (Kanlink.Step = 200);

		CASE Kanlink.Step OF

			0: //nix tun

			100: // Error nr in Logger eintragen

				Kanlink.Step := 200;

			200: // Auf User warten

			1: // init

				Kanlink.KLLib_Init_0(enable := 1, adrServer := ADR(Kanlink),adrInterface := ADR(IFhlKanLink));
				IF Kanlink.KLLib_Init_0.status = ERR_OK THEN
					Kanlink.Step := 10;
				ELSIF Kanlink.KLLib_Init_0.status <> ERR_FUB_BUSY THEN // fehler
					WL_ErrorNr := 10;
					Kanlink.Step := 100;

					IF _xRBReady THEN

						_LogEntryIn.wErrorNo := 10;
						_InsertRB(wPtrStart := _wPtrRBstart, wPtrRead := _wPtrRBread, wPtrWrite := _wPtrRBwrite);

					END_IF

				END_IF;

			10: // Kanlink Run

			20: // Kanlink schliessen

				Kanlink.udp.close.enable := 1;
				Kanlink.udp.close.ident := Kanlink._uiLastId;
				Kanlink.udp.close;
				IF Kanlink.udp.close.status = 0 THEN
					Kanlink.Step := 0;
				ELSIF Kanlink.udp.close.status = ERR_FUB_BUSY THEN

				ELSE
					Kanlink.Step := 100;
				END_IF;

		END_CASE;

		// interne Zustände auf out Struktur legen
		IFhlKanLink.out.iStep  := Kanlink.Step;
		// noch auzufüllen ....
//		IFhlKanLink.out.iError := ??;
//		IFhlKanLink.out.iClientError[0] := ??;
//		IFhlKanLink.out.iServerError[0] := ??;

		// hier beenden wenn zyklus nicht erlaubt
		IF  Kanlink.Step <> 10 THEN
			RETURN;
		END_IF;

		Kanlink;

		// falls Kanlink nix zu tun hat, hier beenden
		IF Kanlink.xReturn THEN
			RETURN;
		END_IF;

		// ------------------------------------------------------------------
		// Falls ein Request eines Clients aufgelaufen ist

		IF Kanlink._xGetServerReq THEN  // Req eines Clients angenommen, bearbeiten

			actGetServerReq;

			Kanlink._xGetServerReq := FALSE;
			Kanlink.udp.rec.enable := 1;

			RETURN;  // Daten sind versendet. Also Ende.

		END_IF;

		// ------------------------------------------------------------------------------
		// falls Response von einem Request kommt:

		IF Kanlink._xGetClientResp THEN // Response auf ClientReq angekommen
			actResponse;

		END_IF;

		// ------------------------------------------------------------------------------
		// Überprüfen ob per Hand bearbeitete Requests versendet werden müssen..

		IF  Kanlink.udp.send.enable = 0 THEN
			_xServerFound := 0;

			FOR _i:=0 TO HLKANLINK_MAX_SERVERCONNS  DO
				_ptrIndex ACCESS ADR(Kanlink.ServerListe[_iLastServerIdx]);
				_dSrvIf ACCESS _ptrIndex.adrInterface;
				IF (_ptrIndex.xReqManually AND (_dSrvIf.iState = 2)) THEN
					_xServerFound := 1;

					_iLastServerIdx := _iLastServerIdx + 1; // testen
					IF _iLastCltIdx > HLKANLINK_MAX_SERVERCONNS THEN
						_iLastServerIdx := 0;
					END_IF;
					EXIT;
					END_IF;
					_iLastServerIdx := _iLastServerIdx + 1; // testen
					IF _iLastServerIdx > HLKANLINK_MAX_SERVERCONNS THEN
					_iLastServerIdx := 0;
				END_IF;

			END_FOR;

			IF _xServerFound THEN
				Kanlink.ServerData.HeaderV1Send[0].Command := _ptrIndex.Cmd + 1;
				Kanlink.ServerData.HeaderV1Send[0].dataFormat := 5;
				Kanlink.ServerData.HeaderV1Send[0].Length := UDINT_TO_UINT( _ptrIndex.RespLength);
				Kanlink.ServerData.HeaderV1Send[0].ReqID := _ptrIndex.iReqID;
				Kanlink.ServerData.HeaderV1Send[0].CmdNr := _ptrIndex.CmdOpt AND 16#00FF;
				_ptrIndex.iConnectionTimer := 0;
				KLLib_SendData(ADR(Kanlink),_ptrIndex.AdrDataResp,_ptrIndex.RespLength,ADR(_ptrIndex.sClientIPAdr),-1,-1,0);
				_dSrvIf.iState := 0;
				RETURN;
			END_IF;
		END_IF;

		IF Kanlink._xSendClient THEN  // hier den Clienten bearbeiten
			_xCltFound := FALSE;
			_iCltIdx := -1;
			_iMuCltIdx := -1;

			FOR _i:=0 TO HLKANLINK_MAX_CLIENTCONNS  DO
				IF (Kanlink.ClientListe[_iLastCltIdx].MuClient >= 0) THEN
					IF ((Kanlink.MuClientListe[Kanlink.ClientListe[_iLastCltIdx].MuClient].bUse = 0) OR (Kanlink.MuClientListe[Kanlink.ClientListe[_iLastCltIdx].MuClient].bUse = 255)) THEN
						_xCheckClt := TRUE;
					ELSE
						_xCheckClt := FALSE;
					END_IF
				ELSE
					_xCheckClt := TRUE;
				END_IF

				IF (_xCheckClt = TRUE) THEN
					_dClient ACCESS ADR(Kanlink.ClientListe[_iLastCltIdx]);
					IF _dClient.adrInterface <> 0 THEN
						_dCltIf ACCESS _dClient.adrInterface;
					ELSE
						_dCltIf ACCESS ADR(_ifDummy);
					END_IF;
						// gefunden wenn kein ReqPend, Commando <> 0 todo gültige Adresse etc...
					IF _dClient.iCycleTime = 0 THEN
						_xSendNow := (_dCltIf.iState = 1) OR (_dCltIf.iState = 4) ; // falls angetickt oder timeout
					ELSE
						_xSendNow := (_dClient.iCycleWait > _dClient.iCycleTime);
					END_IF;
					IF 	(NOT _dClient.xReqPending) AND (_dClient.Cmd <> 0) AND _dClient.xActiv AND (_xSendNow) THEN
			  			_xCltFound := TRUE;
						_iCltIdx := _iLastCltIdx;
						_iLastCltIdx := _iLastCltIdx + 1; // testen
						IF _iLastCltIdx > HLKANLINK_MAX_CLIENTCONNS THEN
				  			_iLastCltIdx := 0;
						END_IF;
						EXIT;
					END_IF;
				END_IF

				_iLastCltIdx := _iLastCltIdx + 1; // testen
				IF _iLastCltIdx > HLKANLINK_MAX_CLIENTCONNS THEN
		  			_iLastCltIdx := 0;
				END_IF;

			END_FOR;

			IF (NOT _xCltFound) THEN
				FOR _i:=0 TO HLKANLINK_MAX_MU_CLIENTCONNS DO
					IF ((Kanlink.MuClientListe[_iLastMuCltIdx].bUse = 1) OR (Kanlink.MuClientListe[_iLastMuCltIdx].bUse = 2)) THEN

						IF Kanlink.ClientListe[Kanlink.MuClientListe[_iLastMuCltIdx].Clients[0]].adrInterface <> 0 THEN
							_dCltIf ACCESS Kanlink.ClientListe[Kanlink.MuClientListe[_iLastMuCltIdx].Clients[0]].adrInterface;
						ELSE
							_dCltIf ACCESS ADR(_ifDummy);
						END_IF;
							// gefunden wenn kein ReqPend, Commando <> 0 todo gültige Adresse etc...
						IF Kanlink.MuClientListe[_iLastMuCltIdx].iCycleTime = 0 THEN
							_xSendNow := (_dCltIf.iState = 1) OR (_dCltIf.iState = 4) ; // falls angetickt oder timeout
						ELSE
							_xSendNow := (Kanlink.MuClientListe[_iLastMuCltIdx].iCycleWait > Kanlink.MuClientListe[_iLastMuCltIdx].iCycleTime);
						END_IF;

						IF 	(NOT Kanlink.MuClientListe[_iLastMuCltIdx].xReqPending) AND Kanlink.MuClientListe[_iLastMuCltIdx].xActiv AND (_xSendNow) THEN
				  			_xCltFound := TRUE;
							_iMuCltIdx := _iLastMuCltIdx;
							_iLastMuCltIdx := _iLastMuCltIdx + 1; // testen
							IF _iLastMuCltIdx > HLKANLINK_MAX_MU_CLIENTCONNS THEN
					  			_iLastMuCltIdx := 0;
							END_IF;
							EXIT;
						END_IF;

					END_IF

					_iLastMuCltIdx := _iLastMuCltIdx + 1; // testen
					IF _iLastMuCltIdx > HLKANLINK_MAX_MU_CLIENTCONNS THEN
			  			_iLastMuCltIdx := 0;
					END_IF;

				END_FOR;
			END_IF

			IF NOT _xCltFound THEN
				Kanlink._xSendClient := FALSE;
				RETURN;

			ELSE

				IF (_iCltIdx >= 0) THEN
					// Client gefunden
					_dClient.iCnt := _dClient.iCnt + 1 ;
					_dClient.iReqId := _dClient.iReqId +1;
					_dClient.TimeOutLeft := _dClient.TimeOut;

					IF _dCltIf.iState = 1 THEN // falls über state dann "schnellwiederholung" aktivieren
						_dClient.iTimeOutCnt := 0; // scharf machen für den nächsten versuch
					END_IF;
					_dCltIf.iState := 2;

					Kanlink.ServerData.HeaderV1Send[0].Command := _dClient.Cmd;
					Kanlink.ServerData.HeaderV1Send[0].CmdNr := _dClient.CmdOpt AND 16#00FF;

					Kanlink.ServerData.HeaderV1Send[0].dataFormat := 5;
					Kanlink.ServerData.HeaderV1Send[0].Length := UDINT_TO_UINT( _dClient.ReqLength);
					Kanlink.ServerData.HeaderV1Send[0].ReqID := _dClient.iReqId;
					Kanlink.ServerData.HeaderV1Send[0].Tag		:= _dCltIf.tag;

// warum ?			KLLib_SendData(ADR(Kanlink),0,                  0,                 ADR(_dClient.sClientAdr),_iCltIdx,-1,KLLIB_REQ);
					KLLib_SendData(ADR(Kanlink),_dClient.AdrDataReq,_dClient.ReqLength,ADR(_dClient.sClientAdr),-1,      -1,KLLIB_REQ);

					_dClient.xReqPending := TRUE;
					_dClient.iCycleWait := 0;

					Kanlink._xSendClient := FALSE;

					RETURN;

				ELSIF (_iMuCltIdx >= 0) THEN

					// Client gefunden
					Kanlink.MuClientListe[_iMuCltIdx].iCnt := Kanlink.MuClientListe[_iMuCltIdx].iCnt + 1;
					Kanlink.MuClientListe[_iMuCltIdx].iReqId := Kanlink.MuClientListe[_iMuCltIdx].iReqId + 1;
					Kanlink.MuClientListe[_iMuCltIdx].TimeOutLeft := Kanlink.MuClientListe[_iMuCltIdx].TimeOut;

					IF _dCltIf.iState = 1 THEN // falls über state dann "schnellwiederholung" aktivieren
						Kanlink.MuClientListe[_iMuCltIdx].iTimeOutCnt := 0; // scharf machen für den nächsten versuch
					END_IF;
					_dCltIf.iState := 2;

					FOR _i := 0 TO KLLIB_MAX_MUL DO

						IF (Kanlink.MuClientListe[_iMuCltIdx].Clients[_i] >= 0) THEN

							Kanlink.ClientListe[Kanlink.MuClientListe[_iMuCltIdx].Clients[_i]].iCnt := Kanlink.MuClientListe[_iMuCltIdx].iCnt;
							Kanlink.ClientListe[Kanlink.MuClientListe[_iMuCltIdx].Clients[_i]].iReqId := Kanlink.MuClientListe[_iMuCltIdx].iReqId;
							Kanlink.ClientListe[Kanlink.MuClientListe[_iMuCltIdx].Clients[_i]].TimeOutLeft := Kanlink.MuClientListe[_iMuCltIdx].TimeOut;

							Kanlink.ServerData.HeaderV1Send[_i].Command := Kanlink.ClientListe[Kanlink.MuClientListe[_iMuCltIdx].Clients[_i]].Cmd;
							Kanlink.ServerData.HeaderV1Send[_i].CmdNr := Kanlink.ClientListe[Kanlink.MuClientListe[_iMuCltIdx].Clients[_i]].CmdOpt AND 16#00FF;

							Kanlink.ServerData.HeaderV1Send[_i].dataFormat := 5;
							Kanlink.ServerData.HeaderV1Send[_i].Length := UDINT_TO_UINT(Kanlink.ClientListe[Kanlink.MuClientListe[_iMuCltIdx].Clients[_i]].ReqLength);
							Kanlink.ServerData.HeaderV1Send[_i].ReqID := Kanlink.ClientListe[Kanlink.MuClientListe[_iMuCltIdx].Clients[_i]].iReqId;
							Kanlink.ServerData.HeaderV1Send[_i].Tag	:= _dCltIf.tag;

						END_IF

					END_FOR

					KLLib_SendData(ADR(Kanlink),0,0,ADR(Kanlink.MuClientListe[_iMuCltIdx].sClientAdr),-1,_iMuCltIdx,KLLIB_REQ);

					Kanlink.MuClientListe[_iMuCltIdx].xReqPending := TRUE;
					Kanlink.MuClientListe[_iMuCltIdx].iCycleWait := 0;

					FOR _i := 0 TO KLLIB_MAX_MUL DO

						IF (Kanlink.MuClientListe[_iMuCltIdx].Clients[_i] >= 0) THEN

							Kanlink.ClientListe[Kanlink.MuClientListe[_iMuCltIdx].Clients[_i]].xReqPending := TRUE;
							Kanlink.ClientListe[Kanlink.MuClientListe[_iMuCltIdx].Clients[_i]].iCycleWait := 0;
						END_IF

					END_FOR

					Kanlink._xSendClient := FALSE;

					RETURN;

				END_IF

			END_IF;

		END_IF;	// sendClient

#ifndef  HLKANLINK_AUTONOM  // wird MIT Framework gearbeitet
	ELSIF IFmnParam.Out.xParamOK AND IFmnEth.Out.xDataValid THEN

		Kanlink.ServerData.MetaInfoResp.KanLink_Hostname := IFmnEth.Out.IP.sHostname;
		Kanlink.ServerData.MetaInfoResp.Machine_type := WSTRING_TO_STRING(IFmnParam.Out.HeaderVersion.utfMachineType);
		Kanlink.ServerData.MetaInfoResp.DataModelTimeStamp := IFmnParam.Out.HeaderVersion.dtTimestamp;
		Kanlink.ServerData.MetaInfoResp.DataModelVersion := IFmnParam.Out.HeaderVersion.wVersion;

		Kanlink.ServerData.PingResp.KanLink_Hostname := IFmnEth.Out.IP.sHostname;

		_xInitOK := TRUE;

	END_IF
#else  // falls OHNE Framework gearbeitet wird
	ELSIF TRUE THEN
		_xInitOK := TRUE;
	END_IF
#endif

END_PROGRAM

PROGRAM _EXIT

	Kanlink.udp.close.enable	:= TRUE;
	Kanlink.udp.close.ident		:= Kanlink.udp.open.ident;
	Kanlink.udp.close;

END_PROGRAM
```

### Library Logical/Standard/Kanlink/KGFramework/Pkg_hlKanLink/KanLinkLib (IEC, version 0.94.5) - KanlinkHilfsfunktionen
Depends on: AsUDP, asstring, AsARCfg, brsystem, sys_lib, AsArLog, AsIODiag, AsETH, DataObj, KL_UserLib, KGstdLib

### KGFramework.ReleaseNotes.txt
```
0.08.0	2012-06-04	- mnParam Version 0.23.0. Siehe history.Pkg_mnParam.txt
					- mnSystem Version 1.04.0. Siehe mnSystem.History.txt
0.09.0	2012-06-12	- mnParam Version 0.24.0. Siehe history.Pkg_mnParam.txt
					- KGStandard Version 1.21.0
					- mnSystem Version 1.05.0
					- svCPCache Version 0.03.0
					- hlDFII Version 1.17.0. ACHTUNG: Parameterstruktur hat sich verändert!!!
0.10.0	2012-06-25	- KGStandar Version 1.22.0
					- mnSystem Version 1.06.0
					- mnParam Version 0.24.1
					- svCPCache Version 0.03.1
0.11.0	2012-07-03	- KGStandard Version 1.23.0
					- mnSystem Version 1.07.0
					- mnMsg Version 1.12.0 - Bugfix
					- mnParam Version 0.24.2 - Bugfix
					- svCPCache Version 0.03.2 - Bugfix
					- mnEth Version 2.10.1 - Bugfix
0.12.0	2012-07-18	- KGStandard Version 1.24.0
0.12.1	2012-08-30	- hlKanLink 0.94.4 - Bugfix
0.12.2	2012-09-03	- mnParam 0.24.3 - Bugfixes
0.13.0	2012-09-04	- mnTxt 0.09.0
					- mnParam 0.25.0
0.14.0	2012-09-05	- mnSystem 1.08.0
					- KGStandard 1.25.0
```

### Package Logical/Standard/Kanlink/KGFrameworkShare - Benutzereinstellungen


### Package Logical/Standard/Kanlink/KGFrameworkShare/Pkg_hlKanLinkUser - Kanlink User

### Library Logical/Standard/Kanlink/KGFrameworkShare/Pkg_hlKanLinkUser/KL_UserLib (IEC, version 0.91.0) - Kanlink User Library

#### KL_UserLib.var - Exported constants
```iecst
(********************************************************************
 * COPYRIGHT -- Herbert Kannegiesser GmbH
 ********************************************************************
 * Library: WL_UserLib
 * File: WL_UserLib.var
 * Author: stahlhut
 * Created: January 10, 2012
 ********************************************************************
 * Constants of library WL_UserLib
 ********************************************************************)
VAR CONSTANT
	HLKANLINK_MAX_CLIENTCONNS : UINT := 10; (*Anzahl der Clienten *)
	HLKANLINK_MAX_SERVERCONNS : UINT := 20; (*Anzahl der Server *)
	HLKANLINK_MAX_MU_CLIENTCONNS : UINT := 5;
	HLKANLINK_MAX_OVERVIEW_DATA : UINT := 35; (*Maximum data transfer on 1 overview connections*)
END_VAR
```


- Library Logical/Standard/Kanlink/KGFrameworkShare/Pkg_mnTestUser/libTestUse (IEC) - Userlibrary für Testadapter (no source held here)

- Program Logical/Standard/Kanlink/KGFrameworkShare/Pkg_mnTestUser/mnTestUser (IEC) - Initialisierung des Test (no source held here)

### Program Logical/Standard/Safety/AccessControl (IEC) - *Mapping to allow access into zones

#### Variables.var
```iecst
VAR
	n : INT;
END_VAR
```

#### Main.st
```iecst
PROGRAM _CYCLIC

//	Std.SafetyOnZone[1]	;High level
//	Std.SafetyOnZone[2]	;Maintenance platform
//	Std.SafetyOnZone[3]	;Low level
//	Std.SafetyOnZone[4]	;Belt load SL's
//	Std.SafetyOnZone[5]	;SSL3
//No access on zone 0

//	SafetyZone[0].BagsInTransit :=  FALSE;  // Safe to enter when false (Switch is NO) FALSE WHEN OK..
//	SafetyZone[0].HoistsOutOfPosition := FALSE; //<-- This is used to stop the door from opening if not position FALSE IS OK -- SWITCH IS NC..

	FOR n := 1 TO MAX_SAFE_ZONES DO
		SafetyZone[n].BagsInTransit :=  FALSE;
	//	SafetyZone[n].HoistsOutOfPosition := Hoist_Safety[n].OutOfPosition;
	END_FOR;

END_PROGRAM
```

### Program Logical/Standard/Safety/Safety (IEC)

#### Variables.var
```iecst
VAR CONSTANT
	MAX_SAFE_SYSTEMS : USINT := 1; (*Number of independant safety systems*)
END_VAR
VAR
	n : UINT;
	transitSettlePT : UDINT; (*Determines the amount of time to wait for bags in transit to settle before opening the interlock*)
	ton_10ms_Transit_Settle : ARRAY[0..MAX_SAFE_ZONES] OF TON_10ms; (*Determines the amount of time to wait for bags in transit to settle before opening the interlock*)
	safeState : ARRAY[0..MAX_SAFE_ZONES] OF USINT; (*USINT that tracks the state of the safe system so it can control the tower light*)
	debounceMasterPT : UDINT;
	masterReset : ARRAY[0..MAX_SAFE_ZONES] OF BOOL;
	ton_10ms_Master_Reset : ARRAY[0..MAX_SAFE_SYSTEMS] OF TON_10ms;
	masterResetRequest : ARRAY[0..MAX_SAFE_SYSTEMS] OF BOOL;
	startUpWarningPT : UDINT;
	ton_10ms_startUp_Warning : ARRAY[0..MAX_SAFE_SYSTEMS] OF TON_10ms;
	tp_10ms_reset_Pulse : TP_10ms;
	enableMasterReset : ARRAY[0..MAX_SAFE_SYSTEMS] OF BOOL;
	ton_10ms_Reset_Debounce : ARRAY[0..MAX_SAFE_ZONES] OF TON_10ms;
	ton_10ms_bagsInTransit : ARRAY[0..MAX_SAFE_ZONES] OF TON_10ms;
	f_trigRequestAccess : ARRAY[0..MAX_SAFE_ZONES] OF F_TRIG;
	ton_entryError : ARRAY[0..MAX_SAFE_ZONES] OF TON_10ms;
	resetRequired : ARRAY[0..MAX_SAFE_SYSTEMS] OF BOOL;
	lockDoor : ARRAY[0..MAX_SAFE_ZONES] OF BOOL;
	tof_HoistsOutOfPosition : ARRAY[0..MAX_SAFE_ZONES] OF TOF_10ms;
	safeZone : REFERENCE TO SafeZoneType;
	startZone : ARRAY[0..MAX_SAFE_SYSTEMS] OF UINT;
	endZone : ARRAY[0..MAX_SAFE_SYSTEMS] OF UINT;
	s : USINT;
	masterZone : BOOL;
	alarmCondition : ARRAY[0..MAX_SAFE_SYSTEMS] OF BOOL;
	tmrAlmOutput : ARRAY[0..MAX_SAFE_SYSTEMS] OF TON;
	masterZoneNo : UINT;
	safe2 : REFERENCE TO SafeZoneType;
END_VAR
```

#### _decodeData.st
```iecst
ACTION _decodeData:

//	Zone Status Encoding
//	0 - Zone Input State
//	1 - Zone Ready FOR Reset
//	2 - E-stop FUB error
//	3 - EDM Input State
//	4 - EDM Ready
//	5 - EDM Error
//	6 - EDM Disabled
//	7 - Zone Dependancy
//	8 - Safe System OK
//	9 - Auto Reset
//	10 - ACCESS Request
//	11 - Zone Status

safeZone.SafeInput				:= safeZone.DataFromSafePLC.0;
safeZone.Zone_Status 			:= safeZone.DataFromSafePLC.11;
safeZone.ResetReady				:= safeZone.DataFromSafePLC.1;
safeZone.RequestAccess		:= safeZone.DataFromSafePLC.10;   // Derived in the PLC from from Zone Healthy and Reset Push button

END_ACTION
```

#### Main.st
```iecst
//---------------------------------------------
//-------------Safety Request------------------
//---------------------------------------------
//V1.00.2 -- 2019 May 24 -- TR -- Fix issue with master reset not working if not ready.
//V1.00.3 -- 2019 June 26 -- TR -- FIx issue with the solenoid not opening if the hoist switch is made after the bagInTransit timers.. Add timer for hoist in position so the hoist cannot be moving past the safe position and open the door.
//V1.00.4 -- 2019 November 11 -- TR -- 	FIX: Issues with the solenoid locking incorrectly,
						//ADD: Control to lift the edge protection gates ( Map Directly to all required outputs.)
//V1.00.5 -- 2020 Decemeber 16 -- TR -- UPDATE : Change to new structure for Safety.
//V1.00.6 -- 2021 January 02 -- TR -- UPDATE : Add Test Mode bit
//V2.00.1 - 2001 Feburary 05 - Change Structures to remove links to direct IO points. Data now comes from Safe PLC.

PROGRAM _INIT

//***************************************************************************************
//	N.B Zone 11 has been faked so we can control the lamp tower correctly FOR the primary
//***************************************************************************************

//DECLARE MAX_SAFE_SYSTEMS IN CONTSTANTS

	startZone[1] := 1;   // Number of the Master Zone
	endZone[1] := 6;	// Last zone in the area
	enableMasterReset[1] := TRUE; // Set to true if master reset is to be used/
//	alarmCondition[1] := system_alarm_1 OR soiled_validation_alarm OR halted;

//	//zone for clean alarms.
//	startZone[2] := 11;   // Number of the Master Zone
//	endZone[2] := MAX_SAFE_ZONES;	// Last zone in the area
//	enableMasterReset[2] := TRUE; // Set to true if master reset is to be used/

	//NB//  A ZONE CANNOT BELONG TO MORE THAN 1 SAFE SYSTEM.

	// MAX Zone if 30

	debounceMasterPT := 476; //4.76 second
	transitSettlePT := 3000; //3000seconds
	startUpWarningPT := 500; //5 secs

	FOR n:=1 TO MAX_SAFE_ZONES DO
		safeState[n] := 4;
	END_FOR;

	#if (MAX_SAFE_ZONES  > 30)
	#error 'Cannot have more than 30 safety zones'
	#endif

END_PROGRAM

PROGRAM _CYCLIC

alarmCondition[1] := system_alarm_1 OR soiled_validation_alarm OR halted;
//alarmCondition[2] := system_alarm_2 OR clean_validation_alarm OR halted;

FOR s := 1 TO MAX_SAFE_SYSTEMS DO

	ton_10ms_startUp_Warning[s].IN:= masterResetRequest[s];
	ton_10ms_startUp_Warning[s].PT:= startUpWarningPT;
	ton_10ms_startUp_Warning[s]();

	IF  ton_10ms_startUp_Warning[s].Q AND Std.Clock1s THEN
		Safety.MasterReset_Comm	:= BIT_SET(Safety.MasterReset_Comm,s);
	ELSE
		Safety.MasterReset_Comm	:= BIT_CLR(Safety.MasterReset_Comm,s);
	END_IF;

	masterZoneNo := startZone[s]; // Number of the master zone for the safe system.

	ton_10ms_Master_Reset[s].IN:= SafetyZone[masterZoneNo].ResetButton AND enableMasterReset[s];//masterResetRequest[s];
	ton_10ms_Master_Reset[s].PT:= debounceMasterPT;
	ton_10ms_Master_Reset[s]();

	IF 	ton_10ms_Master_Reset[s].Q THEN
		masterResetRequest[s] := 1;
	END_IF;

	tmrAlmOutput[s].IN := alarmCondition[s];
	tmrAlmOutput[s].PT := T#5s;
	tmrAlmOutput[s]();

	FOR n:= startZone[s] TO endZone[s] DO

		IF startZone[s] = 0 THEN
			EXIT;
		END_IF;

		safeZone ACCESS ADR(SafetyZone[n]);
		masterZone := (n = startZone[s]);
			safe2 ACCESS ADR(SafetyZone[2]);
		_decodeData;

		//Set the EDM bit//
		IF safeZone.EDM THEN
			Safety.EDM_Comm := BIT_SET(Safety.EDM_Comm,n);
		ELSE
			Safety.EDM_Comm := BIT_CLR(Safety.EDM_Comm,n);
		END_IF;

		//set the reset bit//
		IF safeZone.ResetButton THEN
			Safety.Reset_Comm := BIT_SET(Safety.Reset_Comm,n);
		ELSE
			Safety.Reset_Comm := BIT_CLR(Safety.Reset_Comm,n);
		END_IF;

		//-------------------------------------------------------
		//---------------------Master-reset----------------------
		//-------------------------------------------------------
		IF Std.TestMode AND (Safety.SFW_Version = 0) THEN
			safeZone.DoorLock 	:= FALSE;
			safeZone.LiftGates 	:= FALSE;
			safeZone.Zone_Status 	:= TRUE;
			safeZone.Disable 		:= FALSE;
			safeZone.HaltSys 		:= NOT(safeZone.Zone_Status AND NOT safeZone.Disable);
		ELSE
			lockDoor[n] := FALSE;

			tof_HoistsOutOfPosition[n].IN := safeZone.HoistsOutOfPosition;
			tof_HoistsOutOfPosition[n].PT := 100;
			tof_HoistsOutOfPosition[n]();

			ton_entryError[n].IN := (safeState[n] = 3);
			ton_entryError[n].PT := 100;
			ton_entryError[n]();

			IF ton_10ms_Master_Reset[s].Q AND NOT safeZone.Zone_Status AND safeZone.ResetReady THEN // only put a zone to reset if it needs it
				masterReset[n] := TRUE; // Set masterReset
				safeState[n] := 10; // Goto master reset state
			END_IF;

			//-------------------------------------------------------
			//------------------END-Master-Reset-END-----------------
			//-------------------------------------------------------

			//-------------------------------------------------------
			//------------------Safety-State-Machine-----------------
			//-------------------------------------------------------

			//Wait for bags to finish moving and hoists to get into position.. Door can be unlocked
			ton_10ms_Transit_Settle[n](IN:= safeZone.AccessRequested AND (safeState[n] = 1), PT:=transitSettlePT);
			IF NOT masterZone THEN
				f_trigRequestAccess[n].CLK:= safeZone.RequestAccess;
				f_trigRequestAccess[n]();
			END_IF;
			CASE safeState[n] OF
				0: //Zone reset do not enter

					// Operator requests access by pressing Access DI for 1 second then releasing
					IF safeZone.AccessRequested THEN
						safeState[n] := 1;
					ELSIF safeZone.Zone_Status AND f_trigRequestAccess[n].Q  THEN//	ELSIF (debounceEdgeNeg[n] OR safeZone.AccessRequested) AND NOT masterReset THEN //Look for falling edge if masterReset not requested
						safeZone.AccessRequested := TRUE; //Reset after unlocking or safe zone goes off
						safeState[n] := 1; //Access has been requested
						masterReset[n] := 0;
						//If zone accessed by override or depedant Zone drops out.
					ELSIF NOT safeZone.Zone_Status AND NOT safeZone.SafeInput THEN //If entered with overide goto state 3
						safeState[n] := 3;
					ELSIF NOT safeZone.Zone_Status AND safeZone.SafeInput THEN //If dependant zone drops out
						safeState[n] := 4;
					END_IF;

				1: //Access has been requested
					//Allow 1 second for moving bags to settle, once ok
					ton_10ms_bagsInTransit[n](IN:=NOT safeZone.BagsInTransit, PT:=100); //buffer the BagsInTransit bool

					//Latch solenoid lock open
					IF ton_10ms_bagsInTransit[n].Q AND safeZone.Disable AND NOT tof_HoistsOutOfPosition[n].Q THEN //Use Disable instead of AccessRequested, to ensure one cyclic check with Disable on to stop BagsInTransit being missed
						//safeZone.LockDoors := TRUE; //Reset after reset pressed and door shut
						safeState[n] := 2; //Safe to enter no bags in transit
					ELSIF ton_10ms_Transit_Settle[n].Q THEN
						//safeZone.LockDoors := NOT tof_HoistsOutOfPosition[n].Q; //Reset after reset pressed and door shut
						safeState[n] := 3; //Waiting time elapsed, enter with caution
					END_IF;

					//If zone accessed by override or depedant Zone drops out.
					IF NOT safeZone.Zone_Status AND NOT safeZone.SafeInput THEN //If entered with overide goto state 3
						safeState[n] := 3;
					ELSIF NOT safeZone.Zone_Status AND safeZone.SafeInput THEN //If dependant zone drops out
						safeState[n] := 4;
					ELSIF safeZone.Zone_Status AND f_trigRequestAccess[n].Q THEN //Cancel the request
						safeZone.AccessRequested := FALSE; //Reset after safe zone goes off
						safeState[n] := 4;
					END_IF;

				2..3: //Zone unlocked
					//Reset access request
					lockDoor[n] := NOT tof_HoistsOutOfPosition[n].Q;

					IF safeZone.AccessRequested AND NOT safeZone.Zone_Status THEN
					//	safeZone.AccessRequested := FALSE; //Reset after safe zone goes off
						IF n = 0 THEN
							safeState[n] := 0; //Zone reset do not enter
						END_IF
					ELSIF safeZone.Zone_Status AND f_trigRequestAccess[n].Q  AND safeZone.AccessRequested THEN //Cancel the request
						safeZone.AccessRequested := FALSE; //Reset after safe zone goes off
						safeState[n] := 4;
					ELSIF safeZone.Zone_Status AND NOT safeZone.AccessRequested THEN // zone has been accessed and reset.
						safeState[n] := 0;
					END_IF;

				4:
					//Reset tower light state only if safety plc feedback ok
					IF safeZone.Zone_Status THEN //Check Safe PLC status
						safeState[n] := 0; //Zone reset do not enter
					END_IF;

				10: // Master reset
					IF (safeZone.Zone_Status OR NOT safeZone.ResetReady) THEN
						safeState[n] := 0;
						masterReset[n] := FALSE;
					END_IF;

			END_CASE;

			//	//Lock solenoid
			//	//ton_10ms_Reset_Debounce[n](IN:=safeZone.Interlock.GS_DI_01_Access_Reset, PT:=debouncePT);
			//	IF (safeZone.Interlock.GS_DI_01_Access_Reset AND (safeState[n] > 1) AND NOT masterReset[n]) THEN
			//		//safeZone.LockDoors := FALSE; //Reset after reset pressed and door shut
			//		safeZone.AccessRequested := FALSE;
			//		safeState[n] := 4; // Check zone status
			//		//		ELSIF masterReset AND NOT safeZone.Zone_Status AND safeZone.ResetReady THEN
			//		//			safeState[n] := 10; // Goto master reset state
			//	END_IF;

			//Set disable to safe zone off or access requested
			safeZone.Disable := safeZone.AccessRequested OR NOT safeZone.Zone_Status;

			//-------------------------------------------------------
			//-------END--------Safety State Machine-------END-------
			//-------------------------------------------------------

			//-------------------------------------------------------
			//---------Set tower light status-&-TV-Indicators--------
			//-------------------------------------------------------
			IF NOT masterZone THEN //Light tower 0 does not need to indicate access state.. It is used on the main cab to indicate alarms. See alarm Task.
				safeZone.TowerLight.TL_DO_Green := safeZone.TowerLight.TL_DO_Yellow := safeZone.TowerLight.TL_DO_Red := safeZone.TowerLight.TL_DO_Sounder := 0;
				CASE safeState[n] OF
					0: //Zone reset do not enter
						safeZone.TowerLight.TL_DO_Green 	:= safeZone.Zone_Status;
						safeZone.TowerLight.TL_DO_Red 		:= NOT safeZone.Zone_Status;
					1: //Access has been requested
						safeZone.TowerLight.TL_DO_Yellow 	:= Std.Clock1s; 	//Means Zone Ok but access requested
						safeZone.TowerLight.TL_DO_Green 	:= safeZone.Zone_Status;
						safeZone.TowerLight.TL_DO_Red 		:= NOT safeZone.Zone_Status;
					2: //Safe to enter no bags in transit and hoists in position
						safeZone.TowerLight.TL_DO_Yellow 	:= TRUE; //Amber & RED steady indicates safe to enter
						safeZone.TowerLight.TL_DO_Green 	:= safeZone.Zone_Status;
						safeZone.TowerLight.TL_DO_Red 		:= TRUE;
					3: //
						safeZone.TowerLight.TL_DO_Yellow 	:= Std.Clock200ms; //Amber/Green Alternate-- Enter with Caution
						safeZone.TowerLight.TL_DO_Sounder 	:= NOT ton_entryError[n].Q; //Short alarm to indicate enter with caution
						safeZone.TowerLight.TL_DO_Green 	:= NOT Std.Clock200ms;
						safeZone.TowerLight.TL_DO_Red 		:= NOT Std.Clock200ms OR safeZone.HoistsOutOfPosition; // If red ight on then fault

					4: //Ready for Reset
						safeZone.TowerLight.TL_DO_Yellow 	:= Std.Clock500ms AND safeZone.ResetReady; //Flash Yellow when ready to be reset
						safeZone.TowerLight.TL_DO_Green 	:= safeZone.Zone_Status;

					10://Master Reset Zone about to start
						safeZone.TowerLight.TL_DO_Sounder := TRUE;
						safeZone.TowerLight.TL_DO_Red := Std.Clock200ms; //Red fast flash indicates zone will reset
				END_CASE;

			ELSE // Master Zone lamp controls
				safeZone.TowerLight.TL_DO_Red 		:= FALSE;
				safeZone.TowerLight.TL_DO_Yellow	:= FALSE;
				safeZone.TowerLight.TL_DO_Green	:= FALSE;

				IF safeZone.HaltSys AND NOT safeZone.ResetReady THEN	//Emergency stop blink red. (State 1)
					safeZone.TowerLight.TL_DO_Red 		:= Std.Clock1s ;
				ELSIF safeZone.HaltSys THEN // Estop waiting for reset  (State 2)
					safeZone.TowerLight.TL_DO_Yellow		:= Std.Clock1s;
				ELSIF alarmCondition[s] THEN //State 10 -- Show Warning Not Fault when alarm is on as other parts might still be running
					safeZone.TowerLight.TL_DO_Yellow 	:= TRUE;
					safeZone.TowerLight.TL_DO_Green	 := TRUE;
				ELSE //Machine Running (State 6)
					safeZone.TowerLight.TL_DO_Green	 := TRUE;
				END_IF;
				safeZone.TowerLight.TL_DO_Sounder := (alarmCondition[s] AND NOT tmrAlmOutput[s].Q);

			END_IF;

			//-------------------------------------------------------------
			//-------END-Set tower light status-&-TV-Indicators-END--------
			//-------------------------------------------------------------

			//Check if the master reset has reset all zones.
			IF (masterReset[n] AND NOT safeZone.Zone_Status) THEN
				resetRequired[s] := 1;
			END_IF;

			safeZone.DoorLock := lockDoor[n];
			safeZone.LiftGates := (safeZone.Zone_Status AND (safeZone.BagsInTransit OR NOT safeZone.AccessRequested)); // Edge protection gates.
			safeZone.HaltSys := NOT(safeZone.Zone_Status AND NOT safeZone.Disable);
		END_IF;

	END_FOR;

	IF NOT resetRequired[s] THEN
		masterResetRequest[s] := 0;
	END_IF;
	resetRequired[s] := 0;

	//Flash reset btn on main cabinet
	IF masterResetRequest[s] THEN // We can do a master reset and not out safe 0 to reset
		SafetyZone[startZone[s]].Main_Lamp := Std.Clock200ms;
	ELSE
		SafetyZone[startZone[s]].Main_Lamp := Std.Clock1s AND NOT SafetyZone[startZone[s]].Zone_Status;
	END_IF;

END_FOR;

END_PROGRAM
```

### Program Logical/Standard/Safety/mappSafety (IEC)

#### _visu.st
```iecst
ACTION _visu:

	brsitoa(MappSafety.State,ADR(sState));
	brsitoa(safetyInfo.Status.SafeOSState,ADR(sSafeOsState));
	brsitoa(safetyInfo.Status.SafeNodesState,ADR(sSafeNodeState));
	brsitoa(safetyInfo.Status.SystemState,ADR(sSystemState));
	brsitoa(safetyInfo.Status.OperationalModeState,ADR(sOperationalModeState));

	MappSafety.Visu.ResetError.Enable := MappSafety.Visu.ResetError.Visible	:=  (MappSafety.State = 200);

	MappSafety.Visu.Transfer.Enable 			:= NOT MappSafety.Commands.Transfer AND (MappSafety.State <= 11);
	MappSafety.Visu.Complete.Enable 			:= NOT MappSafety.Commands.Complete AND (MappSafety.State <= 10);
	MappSafety.Visu.ActivateSetupMode.Enable 	:= NOT MappSafety.Commands.ActivateSetupMode AND (MappSafety.State <= 10);
	MappSafety.Visu.Exchange.Enable 			:= NOT MappSafety.Commands.Exchange AND (MappSafety.State <= 10);
	MappSafety.Visu.Format.Enable 				:= NOT MappSafety.Commands.Format AND (MappSafety.State <= 11);
	MappSafety.Visu.Restart.Enable 				:= NOT MappSafety.Commands.Restart AND (MappSafety.State <= 10);

	MappSafety.Visu.Exchange.Visible 	:= MappSafety.Visu.ActivateSetupMode.Visible := safeInfoValid AND NOT safetyInfo.Status.SetupModeActive AND (MappSafety.State <= 10);
	MappSafety.Visu.Transfer.Visible 	:= safeInfoValid AND NOT safetyInfo.SafeApplication.ExistOnSafeLogic;
	MappSafety.Visu.Complete.Visible 	:= safeInfoValid AND (safetyInfo.SafeApplication.ExistOnSafeLogic AND NOT safetyInfo.SafeApplication.Acknowledged) OR safetyInfo.Status.SetupModeActive ;
	MappSafety.Visu.Restart.Visible 	:= 	TRUE;
	MappSafety.Visu.Format.Visible 		:= safeInfoValid;// AND safetyInfo.SafeApplication.ExistOnSafeLogic;

END_ACTION
```

### Program Logical/Standard/Safety/EvueSafety (IEC, version 2.00.1)

#### Main.st - Safet Task must come after all task with gaurded areas
```iecst
//---------------------------------------------
//-------------Safety Request------------------
//---------------------------------------------
//V1.00.2 -- 2019 May 24 -- TR -- Fix issue with master reset not working if not ready.
//V1.00.3 -- 2019 June 26 -- TR -- FIx issue with the solenoid not opening if the hoist switch is made after the bagInTransit timers.. Add timer for hoist in position so the hoist cannot be moving past the safe position and open the door.
//V1.00.4 -- 2019 November 11 -- TR -- 	FIX: Issues with the solenoid locking incorrectly,
						//ADD: Control to lift the edge protection gates ( Map Directly to all required outputs.)
//V1.00.5 -- 2020 Decemeber 16 -- TR -- UPDATE : Change to new structure for Safety.
//V1.00.6 -- 2021 January 02 -- TR -- UPDATE : Add Test Mode bit
//V2.00.1 - 2001 Feburary 05 - Change Structures to remove links to direct IO points. Data now comes from Safe PLC.

PROGRAM _INIT

//***************************************************************************************
//	N.B Zone 11 has been faked so we can control the lamp tower correctly FOR the primary
//***************************************************************************************

//DECLARE MAX_SAFE_SYSTEMS IN CONTSTANTS

	startZone[1] := 0;   // Number of the Master Zone
	endZone[1] := 6;	// Last zone in the area
	enableMasterReset[1] := TRUE; // Set to true if master reset is to be used/
//	alarmCondition[1] := system_alarm_1 OR soiled_validation_alarm OR halted;

//	//zone for clean alarms.
//	startZone[2] := 11;   // Number of the Master Zone
//	endZone[2] := MAX_SAFE_ZONES;	// Last zone in the area
//	enableMasterReset[2] := TRUE; // Set to true if master reset is to be used/

	//NB//  A ZONE CANNOT BELONG TO MORE THAN 1 SAFE SYSTEM.

	// MAX Zone if 30

	debounceMasterPT := 476; //4.76 second
	transitSettlePT := 3000; //3000seconds
	startUpWarningPT := 500; //5 secs

	FOR n:=1 TO MAX_SAFE_ZONES DO
		safeState[n] := 4;
	END_FOR;

	#if (MAX_SAFE_ZONES  > 30)
	#error 'Cannot have more than 30 safety zones'
	#endif

END_PROGRAM

PROGRAM _CYCLIC

alarmCondition[1] := system_alarm_1 OR soiled_validation_alarm OR halted;
//alarmCondition[2] := system_alarm_2 OR clean_validation_alarm OR halted;

FOR s := 1 TO MAX_SAFE_SYSTEMS DO

	ton_10ms_startUp_Warning[s].IN:= masterResetRequest[s];
	ton_10ms_startUp_Warning[s].PT:= startUpWarningPT;
	ton_10ms_startUp_Warning[s]();

	IF  ton_10ms_startUp_Warning[s].Q AND Std.Clock1s THEN
		Safety.MasterReset_Comm	:= BIT_SET(Safety.MasterReset_Comm,s);
	ELSE
		Safety.MasterReset_Comm	:= BIT_CLR(Safety.MasterReset_Comm,s);
	END_IF;

	masterZoneNo := startZone[s]; // Number of the master zone for the safe system.

	ton_10ms_Master_Reset[s].IN:= SafetyZone[masterZoneNo].ResetButton AND enableMasterReset[s];//masterResetRequest[s];
	ton_10ms_Master_Reset[s].PT:= debounceMasterPT;
	ton_10ms_Master_Reset[s]();

	IF 	ton_10ms_Master_Reset[s].Q THEN
		masterResetRequest[s] := 1;
	END_IF;

	tmrAlmOutput[s].IN := alarmCondition[s];
	tmrAlmOutput[s].PT := T#5s;
	tmrAlmOutput[s]();

	FOR n:= startZone[s] TO endZone[s] DO

	//	IF startZone[s] = 0 THEN
	//		EXIT;
	//	END_IF;

		safeZone ACCESS ADR(SafetyZone[n]);
		masterZone := (n = startZone[s]);
			safe2 ACCESS ADR(SafetyZone[2]);
	//	_decodeData;

		//Set the EDM bit//
		IF safeZone.EDM THEN
			Safety.EDM_Comm := BIT_SET(Safety.EDM_Comm,n);
		ELSE
			Safety.EDM_Comm := BIT_CLR(Safety.EDM_Comm,n);
		END_IF;

		//set the reset bit//
		IF safeZone.ResetButton THEN
			Safety.Reset_Comm := BIT_SET(Safety.Reset_Comm,n);
		ELSE
			Safety.Reset_Comm := BIT_CLR(Safety.Reset_Comm,n);
		END_IF;

		//-------------------------------------------------------
		//---------------------Master-reset----------------------
		//-------------------------------------------------------
		IF Std.TestMode AND (Safety.SFW_Version = 0) THEN
			safeZone.DoorLock 	:= FALSE;
			safeZone.LiftGates 	:= FALSE;
			safeZone.Zone_Status 	:= TRUE;
			safeZone.Disable 		:= FALSE;
			safeZone.HaltSys 		:= NOT(safeZone.Zone_Status AND NOT safeZone.Disable);
		ELSE
			lockDoor[n] := FALSE;

			tof_HoistsOutOfPosition[n].IN := safeZone.HoistsOutOfPosition;
			tof_HoistsOutOfPosition[n].PT := 100;
			tof_HoistsOutOfPosition[n]();

			ton_entryError[n].IN := (safeState[n] = 3);
			ton_entryError[n].PT := 100;
			ton_entryError[n]();

			IF ton_10ms_Master_Reset[s].Q AND NOT safeZone.Zone_Status AND safeZone.ResetReady THEN // only put a zone to reset if it needs it
				masterReset[n] := TRUE; // Set masterReset
				safeState[n] := 10; // Goto master reset state
			END_IF;

			//-------------------------------------------------------
			//------------------END-Master-Reset-END-----------------
			//-------------------------------------------------------

			//-------------------------------------------------------
			//------------------Safety-State-Machine-----------------
			//-------------------------------------------------------

			//Wait for bags to finish moving and hoists to get into position.. Door can be unlocked
			ton_10ms_Transit_Settle[n](IN:= safeZone.AccessRequested AND (safeState[n] = 1), PT:=transitSettlePT);
			IF NOT masterZone THEN
				f_trigRequestAccess[n].CLK:= safeZone.RequestAccess;
				f_trigRequestAccess[n]();
			END_IF;
			CASE safeState[n] OF
				0: //Zone reset do not enter

					// Operator requests access by pressing Access DI for 1 second then releasing
					IF safeZone.AccessRequested THEN
						safeState[n] := 1;
					ELSIF safeZone.Zone_Status AND f_trigRequestAccess[n].Q  THEN//	ELSIF (debounceEdgeNeg[n] OR safeZone.AccessRequested) AND NOT masterReset THEN //Look for falling edge if masterReset not requested
						safeZone.AccessRequested := TRUE; //Reset after unlocking or safe zone goes off
						safeState[n] := 1; //Access has been requested
						masterReset[n] := 0;
						//If zone accessed by override or depedant Zone drops out.
					ELSIF NOT safeZone.Zone_Status AND NOT safeZone.SafeInput THEN //If entered with overide goto state 3
						safeState[n] := 3;
					ELSIF NOT safeZone.Zone_Status AND safeZone.SafeInput THEN //If dependant zone drops out
						safeState[n] := 4;
					END_IF;

				1: //Access has been requested
					//Allow 1 second for moving bags to settle, once ok
					ton_10ms_bagsInTransit[n](IN:=NOT safeZone.BagsInTransit, PT:=100); //buffer the BagsInTransit bool

					//Latch solenoid lock open
					IF ton_10ms_bagsInTransit[n].Q AND safeZone.Disable AND NOT tof_HoistsOutOfPosition[n].Q THEN //Use Disable instead of AccessRequested, to ensure one cyclic check with Disable on to stop BagsInTransit being missed
						//safeZone.LockDoors := TRUE; //Reset after reset pressed and door shut
						safeState[n] := 2; //Safe to enter no bags in transit
					ELSIF ton_10ms_Transit_Settle[n].Q THEN
						//safeZone.LockDoors := NOT tof_HoistsOutOfPosition[n].Q; //Reset after reset pressed and door shut
						safeState[n] := 3; //Waiting time elapsed, enter with caution
					END_IF;

					//If zone accessed by override or depedant Zone drops out.
					IF NOT safeZone.Zone_Status AND NOT safeZone.SafeInput THEN //If entered with overide goto state 3
						safeState[n] := 3;
					ELSIF NOT safeZone.Zone_Status AND safeZone.SafeInput THEN //If dependant zone drops out
						safeState[n] := 4;
					ELSIF safeZone.Zone_Status AND f_trigRequestAccess[n].Q THEN //Cancel the request
						safeZone.AccessRequested := FALSE; //Reset after safe zone goes off
						safeState[n] := 4;
					END_IF;

				2..3: //Zone unlocked
					//Reset access request
					lockDoor[n] := NOT tof_HoistsOutOfPosition[n].Q;

					IF safeZone.AccessRequested AND NOT safeZone.Zone_Status THEN
					//	safeZone.AccessRequested := FALSE; //Reset after safe zone goes off
						IF n = 0 THEN
							safeState[n] := 0; //Zone reset do not enter
						END_IF
					ELSIF safeZone.Zone_Status AND f_trigRequestAccess[n].Q  AND safeZone.AccessRequested THEN //Cancel the request
						safeZone.AccessRequested := FALSE; //Reset after safe zone goes off
						safeState[n] := 4;
					ELSIF safeZone.Zone_Status AND NOT safeZone.AccessRequested THEN // zone has been accessed and reset.
						safeState[n] := 0;
					END_IF;

				4:
					//Reset tower light state only if safety plc feedback ok
					IF safeZone.Zone_Status THEN //Check Safe PLC status
						safeState[n] := 0; //Zone reset do not enter
					END_IF;

				10: // Master reset
					IF (safeZone.Zone_Status OR NOT safeZone.ResetReady) THEN
						safeState[n] := 0;
						masterReset[n] := FALSE;
					END_IF;

			END_CASE;

			//	//Lock solenoid
			//	//ton_10ms_Reset_Debounce[n](IN:=safeZone.Interlock.GS_DI_01_Access_Reset, PT:=debouncePT);
			//	IF (safeZone.Interlock.GS_DI_01_Access_Reset AND (safeState[n] > 1) AND NOT masterReset[n]) THEN
			//		//safeZone.LockDoors := FALSE; //Reset after reset pressed and door shut
			//		safeZone.AccessRequested := FALSE;
			//		safeState[n] := 4; // Check zone status
			//		//		ELSIF masterReset AND NOT safeZone.Zone_Status AND safeZone.ResetReady THEN
			//		//			safeState[n] := 10; // Goto master reset state
			//	END_IF;

			//Set disable to safe zone off or access requested
			safeZone.Disable := safeZone.AccessRequested OR NOT safeZone.Zone_Status;

			//-------------------------------------------------------
			//-------END--------Safety State Machine-------END-------
			//-------------------------------------------------------

			//-------------------------------------------------------
			//---------Set tower light status-&-TV-Indicators--------
			//-------------------------------------------------------
			IF NOT masterZone THEN //Light tower 0 does not need to indicate access state.. It is used on the main cab to indicate alarms. See alarm Task.
				safeZone.TowerLight.TL_DO_Green := safeZone.TowerLight.TL_DO_Yellow := safeZone.TowerLight.TL_DO_Red := safeZone.TowerLight.TL_DO_Sounder := 0;
				CASE safeState[n] OF
					0: //Zone reset do not enter
						safeZone.TowerLight.TL_DO_Green 	:= safeZone.Zone_Status;
						safeZone.TowerLight.TL_DO_Red 		:= NOT safeZone.Zone_Status;
					1: //Access has been requested
						safeZone.TowerLight.TL_DO_Yellow 	:= Std.Clock1s; 	//Means Zone Ok but access requested
						safeZone.TowerLight.TL_DO_Green 	:= safeZone.Zone_Status;
						safeZone.TowerLight.TL_DO_Red 		:= NOT safeZone.Zone_Status;
					2: //Safe to enter no bags in transit and hoists in position
						safeZone.TowerLight.TL_DO_Yellow 	:= TRUE; //Amber & RED steady indicates safe to enter
						safeZone.TowerLight.TL_DO_Green 	:= safeZone.Zone_Status;
						safeZone.TowerLight.TL_DO_Red 		:= TRUE;
					3: //
						safeZone.TowerLight.TL_DO_Yellow 	:= Std.Clock200ms; //Amber/Green Alternate-- Enter with Caution
						safeZone.TowerLight.TL_DO_Sounder 	:= NOT ton_entryError[n].Q; //Short alarm to indicate enter with caution
						safeZone.TowerLight.TL_DO_Green 	:= NOT Std.Clock200ms;
						safeZone.TowerLight.TL_DO_Red 		:= NOT Std.Clock200ms OR safeZone.HoistsOutOfPosition; // If red ight on then fault

					4: //Ready for Reset
						safeZone.TowerLight.TL_DO_Yellow 	:= Std.Clock500ms AND safeZone.ResetReady; //Flash Yellow when ready to be reset
						safeZone.TowerLight.TL_DO_Green 	:= safeZone.Zone_Status;

					10://Master Reset Zone about to start
						safeZone.TowerLight.TL_DO_Sounder := TRUE;
						safeZone.TowerLight.TL_DO_Red := Std.Clock200ms; //Red fast flash indicates zone will reset
				END_CASE;

			ELSE // Master Zone lamp controls
				safeZone.TowerLight.TL_DO_Red 		:= FALSE;
				safeZone.TowerLight.TL_DO_Yellow	:= FALSE;
				safeZone.TowerLight.TL_DO_Green	:= FALSE;

				IF safeZone.HaltSys AND NOT safeZone.ResetReady THEN	//Emergency stop blink red. (State 1)
					safeZone.TowerLight.TL_DO_Red 		:= Std.Clock1s ;
				ELSIF safeZone.HaltSys THEN // Estop waiting for reset  (State 2)
					safeZone.TowerLight.TL_DO_Yellow		:= Std.Clock1s;
				ELSIF alarmCondition[s] THEN //State 10 -- Show Warning Not Fault when alarm is on as other parts might still be running
					safeZone.TowerLight.TL_DO_Yellow 	:= TRUE;
					safeZone.TowerLight.TL_DO_Green	 := TRUE;
				ELSE //Machine Running (State 6)
					safeZone.TowerLight.TL_DO_Green	 := TRUE;
				END_IF;
				safeZone.TowerLight.TL_DO_Sounder := (alarmCondition[s] AND NOT tmrAlmOutput[s].Q);

			END_IF;

			//-------------------------------------------------------------
			//-------END-Set tower light status-&-TV-Indicators-END--------
			//-------------------------------------------------------------

			//Check if the master reset has reset all zones.
			IF (masterReset[n] AND NOT safeZone.Zone_Status) THEN
				resetRequired[s] := 1;
			END_IF;

			safeZone.DoorLock := lockDoor[n];
			safeZone.LiftGates := (safeZone.Zone_Status AND (safeZone.BagsInTransit OR NOT safeZone.AccessRequested)); // Edge protection gates.
			safeZone.HaltSys := NOT(safeZone.Zone_Status AND NOT safeZone.Disable);
		END_IF;

	END_FOR;

	IF NOT resetRequired[s] THEN
		masterResetRequest[s] := 0;
	END_IF;
	resetRequired[s] := 0;

	//Flash reset btn on main cabinet
	IF masterResetRequest[s] THEN // We can do a master reset and not out safe 0 to reset
		SafetyZone[startZone[s]].Main_Lamp := Std.Clock200ms;
	ELSE
		SafetyZone[startZone[s]].Main_Lamp := Std.Clock1s AND NOT SafetyZone[startZone[s]].Zone_Status;
	END_IF;

END_FOR;

END_PROGRAM
```

### Program Logical/Standard/Safety/SafetyUI (IEC, version 1.00.1)

#### SafetyUI.st - Implementation code
```iecst
(********************************************************************
* COPYRIGHT -- Bernecker + Rainer
********************************************************************
* Program: SafetySample
* File: SafetySample.st
* Author: B&R
********************************************************************
* Implementation of program SafetySample
********************************************************************
V1.00.1: TR 16/12/20: Clean up task, Add automatic detection OF EPL path AND node. New Structure TO Safety Vars
*)

PROGRAM _INIT

(* command structure for remote control FUB *)
	remotecmd.Version := safeVERSION_R107;	(* version *)
	remotecmd.Password := 'safeplc';				(* password *)
	remotecmd.NewPassword 	:= 'safeplc';

	remoteCmdGetStatus 		:= remotecmd;
	remoteCmdGetStatus.Command		:= safeCMD_STATUS;
	remoteCmdGetStatus.Data			:= 0;
	remoteCmdGetStatus.Number := 10;// ID to show request from auto refresh

	remoteControlcmd ACCESS ADR(remoteCmdGetStatus);

	(* command structure for application download *)
	appcmd1.Version := safeVERSION_R107;	(* version *)
	appcmd1.Password := 'safeplc';					(* password *)
	appcmd1.ApplicationID := 1;				(* application id *)

	(* hide elements in visualization *)
	FOR xcnt := 0 TO SIZEOF(statusButtonActiv) - 1 DO
		statusButtonActiv[xcnt] := 1;
	END_FOR

	(* hide elements in visualization *)
	statusButtonUnlockApp := 1;
	statusButtonUnlockData := 1;
	statusAcknInfoData := 1;
	statusButtonUnlockExtData := 1;
	statusAcknInfoExtData := 1;
	statusDialog := 1;

	(* set SafeLOGIC ID *)
	visuUsedSLIDRemote := 1;
	visuUsedSLIDData := 1;

	slxused := 0;
	safety := 0;
	visuEnableButtons := 0;

END_PROGRAM

PROGRAM _CYCLIC

	//on init make sure we have set the password..
	safePLC_Ok := (Safety.ModuleID  > 0);

	ton_refreshStatus(IN := (safety > 0) AND safePLC_Ok AND NOT safeRemoteControl_0.Busy AND NOT ton_refreshStatus.Q, PT:=100);

//	//Alarm for Hoist
//	IF (safeLogicStatus.SafeOSState <> 16#66) THEN //16# is Run[SAFE]
//		MpAlarmXSet(gAlarmXCore_Link,'SafetyPLCNotRunning');
//	ELSIF EDGEPOS(safeLogicStatus.SafeOSState = 16#66) THEN
//		MpAlarmXReset(gAlarmXCore_Link,'SafetyPLCNotRunning');
//	END_IF;
//	//End of Alarm

	CASE safety OF
		0:// Get nodes and interface info
			getNode.enable := 1;
			getNode.pvName := 'Safety.MasterReset';
			IF (getNode.status = ERR_OK) THEN
				Node := getNode.NodeNumber;
				Interface := getNode.IF_Adr;
				getNode.enable := 0;
				safety := 2;
			ELSIF (getNode.status <> ERR_FUB_BUSY) AND (getNode.status <> ERR_FUB_ENABLE_FALSE)  THEN
				safety := 100;
			END_IF;
			getNode();

		2:// Check the hardware variant
			CASE Safety.ModuleID OF
				16#0000_DD61: //X20SL8100
					slxused := 0;
					safety := 3;

				16#0000_C5B0: // X20 SLX210
				slxused := 1;
				safety := 3;

			END_CASE;

		3: // Set the password on app load
			visuEnableButtons := 0;
			IF safePLC_Ok THEN
				remotecmd.Command 	:= safeCMD_ENTER;
				remotecmd.Number 	:= 0;
				remotecmd.Data		:= safeCMD_SK_PW;
				IF safeRemoteControl_0.Done THEN
					safety := 10;
				ELSIF EDGEPOS(safeRemoteControl_0.Error) THEN
					execute := 0;
				END_IF;
				safeRemoteControl_0(SafeLOGICID := visuUsedSLIDRemote, Execute := execute, pCommandData := ADR(remotecmd));
				execute := 1;
			END_IF;

		10:// RUN UI

			//Lock the control buttons when the fub's are busy.
			visuEnableButtons := safePLC_Ok AND ((remoteControlcmd.Number = 10) OR NOT safeRemoteControl_0.Busy) AND NOT safeDownloadApplication_0.Busy;
			(****************************************************************************************************************************************)
			(****************************************************************************************************************************************)
			(****************************************************************************************************************************************)
			(* show dialog to ackn command *)
			IF (dialogRemoteCmd = 1) THEN
				statusDialog := 0;
				dialogRemoteCmd := 0;
				indexButtonLeft := 0;
				indexButtonRight := 1;
				indexHeaderText := 0;
				IF (remotecmd.Data = safeCMD_SK_FORMAT) THEN
					indexMessageText := 0;
				ELSIF (remotecmd.Data = safeCMD_SK_XCHG) THEN
					indexMessageText := 1;
				ELSIF (remotecmd.Data = safeCMD_1_UDID_ACKN) THEN
					indexMessageText := 2;
				ELSIF (remotecmd.Data = safeCMD_2_UDID_ACKN) THEN
					indexMessageText := 3;
				ELSIF (remotecmd.Data = safeCMD_3_UDID_ACKN) THEN
					indexMessageText := 4;
				ELSIF (remotecmd.Data = safeCMD_4_UDID_ACKN) THEN
					indexMessageText := 5;
				ELSIF (remotecmd.Data =  safeCMD_N_UDID_ACKN) THEN
					indexMessageText := 6;
				ELSIF (remotecmd.Data =  safeCMD_CLEAR_DATA) THEN
					indexMessageText := 7;
				ELSIF (remotecmd.Data = safeCMD_FW_ACKN) THEN
					indexMessageText := 8;
				ELSIF (remotecmd.Data = safeCMD_RESET) THEN
					indexMessageText := 9;
				END_IF
			END_IF

			(* if dialog is ackn execute fub *)
			IF (dialogButtonLeft = 1 AND indexHeaderText = 0) THEN
				executeRemoteCmd := 1;
				dialogButtonLeft := 0;
				statusDialog := 1;
			ELSIF (dialogButtonRight = 1 AND indexHeaderText = 0) THEN
				dialogButtonRight := 0;
				statusDialog := 1;
			END_IF

			(* password must be at least 6 characters long *)
			IF brsstrlen(ADR(remotecmd.NewPassword)) < 6 THEN
				statusSetPassword := 2;
			ELSE
				statusSetPassword := 0;
			END_IF

			IF NOT safeRemoteControl_0.Busy THEN
				IF executeRemoteCmd THEN
					remoteControlcmd ACCESS ADR(remotecmd);
					executeRemoteControl := 1;
					executeRemoteCmd := 0;
				ELSIF ton_refreshStatus.Q THEN  // Set default, so we always read the status cyclically..
					executeRemoteControl := 1;
					remoteControlcmd ACCESS ADR(remoteCmdGetStatus);
				END_IF;
			END_IF;

			safeRemoteControl_0(SafeLOGICID := visuUsedSLIDRemote, Execute := executeRemoteControl, pCommandData := ADR(remoteControlcmd));
			executeRemoteControl := 0; // Make sure we always look at Rising edge inputs.

			(* reset execution flag *)
			IF (safeRemoteControl_0.Done = 1) THEN
				// If we have formatted or reset the key then wait for the PLC
				IF (remoteControlcmd.Data = safeCMD_CLEAR_DATA) OR (remoteControlcmd.Data = safeCMD_SK_FORMAT) THEN
					safety := 0;
				END_IF;
				safeLogicStatus := safeRemoteControl_0.SafeLOGICStatus;
			ELSIF (safeRemoteControl_0.Error = 1) THEN
				safety := 0;
			END_IF

			(* variables for visualization *)
			IF (safeLogicStatus.SafeKEYChanged = 1) THEN
				FOR xcnt := 0 TO SIZEOF(statusButtonActiv) - 1 DO
					statusButtonActiv[xcnt] := 1;
					statusButtonInactiv[xcnt] := 0;
				END_FOR
				statusButtonActiv[1] := 0;
				statusButtonInactiv[1] := 1;
			ELSIF (safeLogicStatus.NumberOfUDIDMismatches = 1 AND safeLogicStatus.Scanning = 0) THEN
				FOR xcnt := 0 TO SIZEOF(statusButtonActiv) - 1 DO
					statusButtonActiv[xcnt] := 1;
					statusButtonInactiv[xcnt] := 0;
				END_FOR
				statusButtonActiv[3] := 0;
				statusButtonInactiv[3] := 1;
			ELSIF (safeLogicStatus.NumberOfUDIDMismatches = 2 AND safeLogicStatus.Scanning = 0) THEN
				FOR xcnt := 0 TO SIZEOF(statusButtonActiv) - 1 DO
					statusButtonActiv[xcnt] := 1;
					statusButtonInactiv[xcnt] := 0;
				END_FOR
				statusButtonActiv[4] := 0;
				statusButtonInactiv[4] := 1;
			ELSIF (safeLogicStatus.NumberOfUDIDMismatches = 3 AND safeLogicStatus.Scanning = 0) THEN
				FOR xcnt := 0 TO SIZEOF(statusButtonActiv) - 1 DO
					statusButtonActiv[xcnt] := 1;
					statusButtonInactiv[xcnt] := 0;
				END_FOR
				statusButtonActiv[5] := 0;
				statusButtonInactiv[5] := 1;
			ELSIF (safeLogicStatus.NumberOfUDIDMismatches = 4 AND safeLogicStatus.Scanning = 0) THEN
				FOR xcnt := 0 TO SIZEOF(statusButtonActiv) - 1 DO
					statusButtonActiv[xcnt] := 1;
					statusButtonInactiv[xcnt] := 0;
				END_FOR
				statusButtonActiv[6] := 0;
				statusButtonInactiv[6] := 1;
			ELSIF (safeLogicStatus.NumberOfUDIDMismatches > 4 AND safeLogicStatus.Scanning = 0) THEN
				FOR xcnt := 0 TO SIZEOF(statusButtonActiv) - 1 DO
					statusButtonActiv[xcnt] := 1;
					statusButtonInactiv[xcnt] := 0;
				END_FOR
				statusButtonActiv[7] := 0;
				statusButtonInactiv[7] := 1;
			ELSIF (safeLogicStatus.NumberOfDifferentFirmware <> 0 AND safeLogicStatus.Scanning = 0) THEN
				FOR xcnt := 0 TO SIZEOF(statusButtonActiv) - 1 DO
					statusButtonActiv[xcnt] := 1;
					statusButtonInactiv[xcnt] := 0;
				END_FOR
				statusButtonActiv[11] := 0;
				statusButtonInactiv[11] := 1;
			ELSE
				FOR xcnt := 0 TO SIZEOF(statusButtonActiv) - 1 DO
					statusButtonActiv[xcnt] := 1;
					statusButtonInactiv[xcnt] := 0;
				END_FOR
			END_IF
			(* status text - MXCHG *)
			IF (safeLogicStatus.LedTestActive = 1) THEN
				indexMxchgLed := 40;
			ELSIF (safeLogicStatus.Scanning = 1) THEN
				indexMxchgLed := 30;
			ELSIF (safeLogicStatus.NumberOfUDIDMismatches = 1) THEN
				indexMxchgLed := 1;
			ELSIF (safeLogicStatus.NumberOfUDIDMismatches = 2) THEN
				indexMxchgLed := 2;
			ELSIF (safeLogicStatus.NumberOfUDIDMismatches = 3) THEN
				indexMxchgLed := 3;
			ELSIF (safeLogicStatus.NumberOfUDIDMismatches = 4) THEN
				indexMxchgLed := 4;
			ELSIF (safeLogicStatus.NumberOfUDIDMismatches > 4) THEN
				indexMxchgLed := 5;
			ELSIF (safeLogicStatus.NumberOfMissingModules <> 0) THEN
				indexMxchgLed := 20;
			ELSIF (safeLogicStatus.NumberOfUDIDMismatches = 0) THEN
				indexMxchgLed := 10;
			END_IF
			(* status text - FW-ACKN *)
			IF (safeLogicStatus.SafeKEYChanged = 0 AND safeLogicStatus.NumberOfDifferentFirmware = 0) THEN
				indexFwAcknLed := 10;
			ELSIF (safeLogicStatus.SafeKEYChanged = 1) THEN
				indexFwAcknLed := 1;
			ELSIF (safeLogicStatus.NumberOfDifferentFirmware <> 0) THEN
				indexFwAcknLed := 2;
			END_IF
			(* status text - FAIL *)
			IF (safeLogicStatus.FailSafe <> 16#55) THEN
				indexFAILLed := 2;
			ELSIF (safeLogicStatus.openSAFETYstate = 0) THEN
				indexFAILLed := 0;
			ELSIF (safeLogicStatus.openSAFETYstate = 1) THEN
				indexFAILLed := 1;
			END_IF
			(* status text - R/E *)
			indexRELed := safeLogicStatus.SafeOSState;

			(****************************************************************************************************************************************)
			(****************************************************************************************************************************************)
			(****************************************************************************************************************************************)
			(* show dialog to ackn command *)
			IF (dialogApplication = 1) THEN
				IF (statusDialog  <> 0) THEN
					statusDialog := 0;
					dialogApplication := 0;
					indexButtonLeft := 0;
					indexButtonRight := 1;
					indexHeaderText := 1;
					indexMessageText := 10;
				ELSE
					statusDialog := 1;
				END_IF;
			END_IF

			(* if dialog is ackn unlock application *)
			IF (dialogButtonLeft = 1 AND indexHeaderText = 1) THEN
				executeapp1 := 1;
				appcmd1.Unlock := 1;
				dialogButtonLeft := 0;
				statusDialog := 1;
			ELSIF (dialogButtonRight = 1 AND indexHeaderText = 1) THEN
				executeapp1 := 1;
				appcmd1.Unlock := 2;
				dialogButtonRight := 0;
				statusDialog := 1;
			END_IF

			(* convert application CRC to HEX string *)
			itoahex(safeDownloadApplication_0.ApplicationCRC, ADR(visuApplicationCRC));

			safeDownloadApplication_0(SafeLOGICID := appcmd1.ApplicationID, Execute := executeapp1, pCommandData := ADR(appcmd1));
			(* show unlock button *)
			IF (safeDownloadApplication_0.UnlockRequired = 1) THEN
				statusButtonUnlockApp := 0;
			ELSE
				appcmd1.Unlock := 0;
				statusButtonUnlockApp := 1;
			END_IF
			IF EDGEPOS(safeDownloadApplication_0.UnlockRequired = 1) THEN
				dialogApplication := 1;
			END_IF;

			IF (safeDownloadApplication_0.Done OR safeDownloadApplication_0.Error)  THEN
				executeapp1 := 0;
			END_IF;

			(* read UDID from SafeLOGIC-X *)
			UDID_Low := Safety.UDID_low;
			UDID_High := Safety.UDID_high;

//			IF slxused = 1 THEN
//				readUDIDlowSLX(enable := 1, pDeviceName := ADR(Station), pChannelName := ADR('UDID_low'));
//
//				IF readUDIDlowSLX.status = 0 THEN
//					UDID_Low := readUDIDlowSLX.value;
//				ELSIF readUDIDlowSLX.status <> 65535 THEN
//					UDID_Low := 0;
//				END_IF
//
//				readUDIDhighSLX(enable := 1, pDeviceName := ADR(Station), pChannelName := ADR('UDID_high'));
//
//				IF readUDIDhighSLX.status = 0 THEN
//					UDID_High := UDINT_TO_UINT(readUDIDhighSLX.value);
//				ELSIF readUDIDhighSLX.status <> 65535 THEN
//					UDID_High := 0;
//				END_IF
//
//				(* hide / show visualization elements *)
//				stautsSLXInformation := 0;
//				statusSLInformation := 1;
//				(* read UDID form SafeLOGIC *)
//			ELSE
//				readUDIDlowSL(enable := 1, pDevice := ADR(Interface), node := Node, index := 16#2000, subindex := 6, pData := ADR(UDID_Low), datalen := SIZEOF(UDID_Low));
//
//				IF readUDIDlowSL.status <> 0 AND readUDIDlowSL.status <> 65535 THEN
//					UDID_Low := 0;
//				END_IF
//
//				readUDIDhighSL(enable := 1, pDevice := ADR(Interface), node := Node, index := 16#2000, subindex := 7, pData := ADR(UDID_High), datalen := SIZEOF(UDID_High));
//
//				IF readUDIDhighSL.status <> 0 AND readUDIDhighSL.status <> 65535 THEN
//					UDID_High := 0;
//				END_IF
//
//				(* hide / show visualization elements *)
//				stautsSLXInformation := 1;
//				statusSLInformation := 0;
//			END_IF

		100://Error

	END_CASE;

	(* convert UDID to HEX string *)
	itoahex(UDID_Low, ADR(visuUDID_Low));
	itoahex(UDID_High, ADR(visuUDID_High));

	(****************************************************************************************************************************************)
	(****************************************************************************************************************************************)
	(****************************************************************************************************************************************)
	(* write UDID for SafeLOGIC to command structure *)
	appcmd1.UDID_Low := UDID_Low;
	appcmd1.UDID_High := UDID_High;
	datacmd1.UDID_Low := UDID_Low;
	datacmd1.UDID_High := UDID_High;
	datacmd2.UDID_Low := UDID_Low;
	datacmd2.UDID_High := UDID_High;

	(****************************************************************************************************************************************)
	(****************************************************************************************************************************************)
	(****************************************************************************************************************************************)
	(* mappView lists use strings for values rather than int,uint etc. convert UINT to Strings. *)
	strRE_Led := UINT_TO_STRING(indexRELed);
	strMXCHG_Led := UINT_TO_STRING(indexMxchgLed);
	strFWACKN_Led := UINT_TO_STRING(indexFwAcknLed);
	strFAIL_Led := UINT_TO_STRING(indexFAILLed);

	IF NOT safePLC_Ok THEN
		strStatusID := '10';
	ELSIF (safety = 0) THEN
		IF (safeRemoteControl_0.StatusID = ERR_FUB_BUSY) THEN
			strStatusID := '11';
		ELSE
			strStatusID := UINT_TO_STRING(safeRemoteControl_0.StatusID);
		END_IF;
	ELSIF safeDownloadApplication_0.Busy OR safeDownloadApplication_0.Error  THEN
		strStatusID := UINT_TO_STRING(safeDownloadApplication_0.StatusID);
	ELSIF  ((safeRemoteControl_0.Busy AND remoteControlcmd.Number <> 10) OR safeRemoteControl_0.Error)  THEN
		strStatusID := UINT_TO_STRING(safeRemoteControl_0.StatusID);
	ELSE
		strStatusID := '1';//NOTHING
	END_IF;

	strStatus := UINT_TO_STRING(safeLogicStatus.Status);

	strDownloadStatus := UINT_TO_STRING(safeDownloadApplication_0.StatusID);
	//strDataStatus := UINT_TO_STRING(safeDownloadData_0.StatusID);
	strMessageTest := UINT_TO_STRING(indexMessageText);

	(* guide user by changing button to orange. *)
	IF (statusButtonActiv[0] = 1) THEN
		strSKFormatStyle := 'Kannegiesser1';
	ELSE
		strSKFormatStyle := 'orange';
	END_IF;

	IF (statusButtonActiv[1] = 1) THEN
		strSKXCHGtStyle := 'Kannegiesser1';
	ELSE
		strSKXCHGtStyle := 'orange';
	END_IF;

	IF (statusButtonActiv[2] = 1) THEN
		strScanStyle := 'Kannegiesser1';
	ELSE
		strScanStyle := 'orange';
	END_IF;

	IF (statusButtonActiv[3] = 1) THEN
		strAck1Style := 'Kannegiesser1';
	ELSE
		strAck1Style := 'orange';
	END_IF;

	IF (statusButtonActiv[4] = 1) THEN
		strAck2Style := 'Kannegiesser1';
	ELSE
		strAck2Style := 'orange';
	END_IF;

	IF (statusButtonActiv[5] = 1) THEN
		strAck3Style := 'Kannegiesser1';
	ELSE
		strAck3Style := 'orange';
	END_IF;

	IF (statusButtonActiv[6] = 1) THEN
		strAck4Style := 'Kannegiesser1';
	ELSE
		strAck4Style := 'orange';
	END_IF;

	IF (statusButtonActiv[7] = 1) THEN
		strAckNStyle := 'Kannegiesser1';
	ELSE
		strAckNStyle := 'orange';
	END_IF;

	IF (statusButtonActiv[8] = 1) THEN
		strClearStyle := 'Kannegiesser1';
	ELSE
		strClearStyle := 'orange';
	END_IF;

	IF (statusButtonActiv[9] = 1) THEN
		strTestStyle := 'Kannegiesser1';
	ELSE
		strTestStyle := 'orange';
	END_IF;

	IF (statusButtonActiv[11] = 1) THEN
		strFWACKNStyle := 'Kannegiesser1';
	ELSE
		strFWACKNStyle := 'orange';
	END_IF;

	IF (statusButtonUnlockApp = 0) THEN
		bVisAppButtons := TRUE;
	ELSE
		bVisAppButtons := FALSE;
	END_IF;

	IF (statusSLInformation = 0) THEN
		bVisInterfaceNode := TRUE;
		bVisStation := FALSE;
	ELSE
		bVisInterfaceNode := FALSE;
		bVisStation := TRUE;
	END_IF;

			END_PROGRAM
```
